LIN {X 0,Y 115.014,Z 337.015,A -85,B 0,C 180,E1 -25713.825,E2 -25713.825} C_VEL
LIN {X 0,Y 114.868,Z 336.176,A -85,B 0,C 180,E1 -25714.155,E2 -25714.155} C_VEL
LIN {X 0,Y 114.957,Z 336.153,A -85,B 0,C 180,E1 -25718.48,E2 -25718.48} C_VEL
LIN {X 0,Y 115.09,Z 336.142,A -85,B 0,C 180,E1 -25725.861,E2 -25725.861} C_VEL
LIN {X 0,Y 115.315,Z 336.105,A -85,B 0,C 180,E1 -25729.464,E2 -25729.464} C_VEL
LIN {X 0,Y 115.522,Z 336.071,A -85,B 0,C 180,E1 -25736.511,E2 -25736.511} C_VEL
LIN {X 0,Y 115.999,Z 336.032,A -85,B 0,C 180,E1 -25739.999,E2 -25739.999} C_VEL
LIN {X 0,Y 115.369,Z 336.065,A -85,B 0,C 180,E1 -25746.997,E2 -25746.997} C_VEL
LIN {X 0,Y 115.214,Z 336.133,A -85,B 0,C 180,E1 -25752.56,E2 -25752.56} C_VEL
LIN {X 0,Y 114.993,Z 336.157,A -85,B 0,C 180,E1 -25757.793,E2 -25757.793} C_VEL
LIN {X 0,Y 114.954,Z 336.155,A -85,B 0,C 180,E1 -25763.488,E2 -25763.488} C_VEL
LIN {X 0,Y 114.864,Z 336.171,A -85,B 0,C 180,E1 -25771.054,E2 -25771.054} C_VEL
LIN {X 0,Y 114.786,Z 336.182,A -85,B 0,C 180,E1 -25777.753,E2 -25777.753} C_VEL
LIN {X 0,Y 114.854,Z 336.215,A -85,B 0,C 180,E1 -25781.569,E2 -25781.569} C_VEL
LIN {X 0,Y 115.591,Z 338.609,A -85,B 0,C 180,E1 -25782.393,E2 -25782.393} C_VEL
LIN {X 0,Y 117.297,Z 340.754,A -85,B 0,C 180,E1 -25783.84,E2 -25783.84} C_VEL
LIN {X 0,Y 118.632,Z 341.83,A -85,B 0,C 180,E1 -25784.849,E2 -25784.849} C_VEL
LIN {X 0,Y 120.483,Z 344.932,A -85,B 0,C 180,E1 -25786.329,E2 -25786.329} C_VEL
LIN {X 0,Y 122.291,Z 346.894,A -85,B 0,C 180,E1 -25787.589,E2 -25787.589} C_VEL
LIN {X 0,Y 128.039,Z 355.27,A -85,B 0,C 180,E1 -25791.345,E2 -25791.345} C_VEL
LIN {X 0,Y 132.282,Z 362.156,A -85,B 0,C 180,E1 -25793.819,E2 -25793.819} C_VEL
LIN {X 0,Y 137.779,Z 372.248,A -85,B 0,C 180,E1 -25796.776,E2 -25796.776} C_VEL
LIN {X 0,Y 142.801,Z 383.272,A -85,B 0,C 180,E1 -25799.292,E2 -25799.292} C_VEL
LIN {X 0,Y 139.384,Z 431.741,A -85,B 0,C 180,E1 -25801.446,E2 -25801.446} C_VEL
LIN {X 0,Y 137.61,Z 444.886,A -85,B 0,C 180,E1 -25802.518,E2 -25802.518} C_VEL
LIN {X 0,Y 135.307,Z 457.913,A -85,B 0,C 180,E1 -25804.21,E2 -25804.21} C_VEL
LIN {X 0,Y 132.086,Z 470.579,A -85,B 0,C 180,E1 -25806.476,E2 -25806.476} C_VEL
LIN {X 0,Y 128.848,Z 481.799,A -85,B 0,C 180,E1 -25809.23,E2 -25809.23} C_VEL
LIN {X 0,Y 125.616,Z 491.287,A -85,B 0,C 180,E1 -25812.226,E2 -25812.226} C_VEL
LIN {X 0,Y 122.323,Z 500.241,A -85,B 0,C 180,E1 -25815.862,E2 -25815.862} C_VEL
LIN {X 0,Y 118.762,Z 509.308,A -85,B 0,C 180,E1 -25820.629,E2 -25820.629} C_VEL
LIN {X 0,Y 116.029,Z 516.6,A -85,B 0,C 180,E1 -25825.653,E2 -25825.653} C_VEL
LIN {X 0,Y 114.373,Z 521.514,A -85,B 0,C 180,E1 -25829.995,E2 -25829.995} C_VEL
LIN {X 0,Y 112.963,Z 526.412,A -85,B 0,C 180,E1 -25835.482,E2 -25835.482} C_VEL
LIN {X 0,Y 112.094,Z 529.991,A -85,B 0,C 180,E1 -25840.836,E2 -25840.836} C_VEL
LIN {X 0,Y 111.893,Z 531.873,A -85,B 0,C 180,E1 -25844.545,E2 -25844.545} C_VEL
LIN {X 0,Y 112.339,Z 533.886,A -85,B 0,C 180,E1 -25850.216,E2 -25850.216} C_VEL
LIN {X 0,Y 113.447,Z 534.9,A -85,B 0,C 180,E1 -25855.693,E2 -25855.693} C_VEL
LIN {X 0,Y 115.8,Z 534.902,A -85,B 0,C 180,E1 -25861.826,E2 -25861.826} C_VEL
LIN {X 0,Y 118.399,Z 534.078,A -85,B 0,C 180,E1 -25866.405,E2 -25866.405} C_VEL
LIN {X 0,Y 122.562,Z 532.001,A -85,B 0,C 180,E1 -25871.803,E2 -25871.803} C_VEL
LIN {X 0,Y 126.828,Z 529.279,A -85,B 0,C 180,E1 -25876.078,E2 -25876.078} C_VEL
LIN {X 0,Y 132.129,Z 525.316,A -85,B 0,C 180,E1 -25880.337,E2 -25880.337} C_VEL
LIN {X 0,Y 138.279,Z 519.935,A -85,B 0,C 180,E1 -25884.401,E2 -25884.401} C_VEL
LIN {X 0,Y 145.281,Z 512.794,A -85,B 0,C 180,E1 -25888.21,E2 -25888.21} C_VEL
LIN {X 0,Y 152.135,Z 504.673,A -85,B 0,C 180,E1 -25891.359,E2 -25891.359} C_VEL
LIN {X 0,Y 158.91,Z 495.272,A -85,B 0,C 180,E1 -25894.011,E2 -25894.011} C_VEL
LIN {X 0,Y 165.11,Z 484.9,A -85,B 0,C 180,E1 -25896.218,E2 -25896.218} C_VEL
LIN {X 0,Y 170.629,Z 473.828,A -85,B 0,C 180,E1 -25897.961,E2 -25897.961} C_VEL
LIN {X 0,Y 175.101,Z 462.431,A -85,B 0,C 180,E1 -25899.328,E2 -25899.328} C_VEL
LIN {X 0,Y 179.002,Z 449.556,A -85,B 0,C 180,E1 -25900.427,E2 -25900.427} C_VEL
LIN {X 0,Y 181.7,Z 436.861,A -85,B 0,C 180,E1 -25901.178,E2 -25901.178} C_VEL
LIN {X 0,Y 183.622,Z 421.119,A -85,B 0,C 180,E1 -25901.708,E2 -25901.708} C_VEL
LIN {X 0,Y 183.896,Z 418.251,A -85,B 0,C 180,E1 -25901.788,E2 -25901.788} C_VEL
LIN {X 0,Y 179.881,Z 410.116,A -85,B 0,C 180,E1 -25905.361,E2 -25905.361} C_VEL
LIN {X 0,Y 175.899,Z 402.879,A -85,B 0,C 180,E1 -25909.643,E2 -25909.643} C_VEL
LIN {X 0,Y 173.679,Z 399.15,A -85,B 0,C 180,E1 -25912.59,E2 -25912.59} C_VEL
LIN {X 0,Y 171.748,Z 395.552,A -85,B 0,C 180,E1 -25915.973,E2 -25915.973} C_VEL
LIN {X 0,Y 169.873,Z 392.584,A -85,B 0,C 180,E1 -25920.642,E2 -25920.642} C_VEL
LIN {X 0,Y 169.52,Z 391.116,A -85,B 0,C 180,E1 -25922.377,E2 -25922.377} C_VEL
LIN {X 0,Y 169.178,Z 391.143,A -85,B 0,C 180,E1 -25930.637,E2 -25930.637} C_VEL
LIN {X 0,Y 169.496,Z 391.694,A -85,B 0,C 180,E1 -25932.335,E2 -25932.335} C_VEL
LIN {X 0,Y 171.097,Z 395.184,A -85,B 0,C 180,E1 -25937.359,E2 -25937.359} C_VEL
LIN {X 0,Y 171.896,Z 396.213,A -85,B 0,C 180,E1 -25938.945,E2 -25938.945} C_VEL
LIN {X 0,Y 174.141,Z 400.931,A -85,B 0,C 180,E1 -25942.76,E2 -25942.76} C_VEL
LIN {X 0,Y 176.288,Z 405.612,A -85,B 0,C 180,E1 -25945.614,E2 -25945.614} C_VEL
LIN {X 0,Y 178.988,Z 412.031,A -85,B 0,C 180,E1 -25948.682,E2 -25948.682} C_VEL
LIN {X 0,Y 181.92,Z 419.645,A -85,B 0,C 180,E1 -25951.582,E2 -25951.582} C_VEL
LIN {X 0,Y 183.373,Z 423.898,A -85,B 0,C 180,E1 -25952.919,E2 -25952.919} C_VEL
LIN {X 0,Y 181.387,Z 441.689,A -85,B 0,C 180,E1 -25953.52,E2 -25953.52} C_VEL
LIN {X 0,Y 178.821,Z 454.037,A -85,B 0,C 180,E1 -25954.137,E2 -25954.137} C_VEL
LIN {X 0,Y 174.995,Z 466.814,A -85,B 0,C 180,E1 -25955.105,E2 -25955.105} C_VEL
LIN {X 0,Y 170.124,Z 478.957,A -85,B 0,C 180,E1 -25956.342,E2 -25956.342} C_VEL
LIN {X 0,Y 164.688,Z 489.87,A -85,B 0,C 180,E1 -25957.87,E2 -25957.87} C_VEL
LIN {X 0,Y 158.183,Z 500.692,A -85,B 0,C 180,E1 -25959.974,E2 -25959.974} C_VEL
LIN {X 0,Y 151.946,Z 509.507,A -85,B 0,C 180,E1 -25962.271,E2 -25962.271} C_VEL
LIN {X 0,Y 144.869,Z 518.154,A -85,B 0,C 180,E1 -25965.303,E2 -25965.303} C_VEL
LIN {X 0,Y 138.224,Z 525.085,A -85,B 0,C 180,E1 -25968.631,E2 -25968.631} C_VEL
LIN {X 0,Y 132.194,Z 530.666,A -85,B 0,C 180,E1 -25972.316,E2 -25972.316} C_VEL
LIN {X 0,Y 126.992,Z 535.081,A -85,B 0,C 180,E1 -25976.404,E2 -25976.404} C_VEL
LIN {X 0,Y 123.881,Z 537.431,A -85,B 0,C 180,E1 -25979.303,E2 -25979.303} C_VEL
LIN {X 0,Y 121.001,Z 539.364,A -85,B 0,C 180,E1 -25982.318,E2 -25982.318} C_VEL
LIN {X 0,Y 118.527,Z 540.877,A -85,B 0,C 180,E1 -25985.483,E2 -25985.483} C_VEL
LIN {X 0,Y 116.404,Z 541.961,A -85,B 0,C 180,E1 -25988.767,E2 -25988.767} C_VEL
LIN {X 0,Y 113.635,Z 543.009,A -85,B 0,C 180,E1 -25995.683,E2 -25995.683} C_VEL
LIN {X 0,Y 112.838,Z 542.97,A -85,B 0,C 180,E1 -25999.236,E2 -25999.236} C_VEL
LIN {X 0,Y 112.422,Z 542.512,A -85,B 0,C 180,E1 -26002.823,E2 -26002.823} C_VEL
LIN {X 0,Y 112.337,Z 541.661,A -85,B 0,C 180,E1 -26006.419,E2 -26006.419} C_VEL
LIN {X 0,Y 112.45,Z 540.411,A -85,B 0,C 180,E1 -26010.005,E2 -26010.005} C_VEL
LIN {X 0,Y 112.324,Z 537.663,A -85,B 0,C 180,E1 -26015.391,E2 -26015.391} C_VEL
LIN {X 0,Y 112.812,Z 533.857,A -85,B 0,C 180,E1 -26020.777,E2 -26020.777} C_VEL
LIN {X 0,Y 113.958,Z 528.881,A -85,B 0,C 180,E1 -26026.118,E2 -26026.118} C_VEL
LIN {X 0,Y 116.11,Z 522.613,A -85,B 0,C 180,E1 -26031.3,E2 -26031.3} C_VEL
LIN {X 0,Y 119.023,Z 514.744,A -85,B 0,C 180,E1 -26036.291,E2 -26036.291} C_VEL
LIN {X 0,Y 121.441,Z 508.027,A -85,B 0,C 180,E1 -26039.69,E2 -26039.69} C_VEL
LIN {X 0,Y 124.527,Z 500.023,A -85,B 0,C 180,E1 -26042.908,E2 -26042.908} C_VEL
LIN {X 0,Y 127.974,Z 489.74,A -85,B 0,C 180,E1 -26046.188,E2 -26046.188} C_VEL
LIN {X 0,Y 128.825,Z 487.057,A -85,B 0,C 180,E1 -26046.906,E2 -26046.906} C_VEL
LIN {X 0,Y 130.77,Z 488.171,A -85,B 0,C 180,E1 -26048.275,E2 -26048.275} C_VEL
LIN {X 0,Y 130.77,Z 550.146,A -85,B 0,C 180,E1 -26048.275,E2 -26048.275} C_VEL
LIN {X 0,Y 112.288,Z 550.146,A -85,B 0,C 180,E1 -26012.241,E2 -26012.241} C_VEL
LIN {X 0,Y 112.475,Z 548.146,A -85,B 0,C 180,E1 -26011.226,E2 -26011.226} C_VEL
LIN {X 0,Y 112.475,Z 542.371,A -85,B 0,C 180,E1 -26011.226,E2 -26011.226} C_VEL
LIN {X 0,Y 112.45,Z 540.411,A -85,B 0,C 180,E1 -26010.005,E2 -26010.005} C_VEL
LIN {X 0,Y 111.781,Z 539.072,A -85,B 0,C 180,E1 -26012.92,E2 -26012.92} C_VEL
LIN {X 0,Y 110.239,Z 537.452,A -85,B 0,C 180,E1 -26015.767,E2 -26015.767} C_VEL
LIN {X 0,Y 106.959,Z 533.382,A -85,B 0,C 180,E1 -26021.49,E2 -26021.49} C_VEL
LIN {X 0,Y 106.435,Z 530.884,A -85,B 0,C 180,E1 -26024.401,E2 -26024.401} C_VEL
LIN {X 0,Y 106.583,Z 529.982,A -85,B 0,C 180,E1 -26025.356,E2 -26025.356} C_VEL
LIN {X 0,Y 109.008,Z 522.962,A -85,B 0,C 180,E1 -26031.765,E2 -26031.765} C_VEL
LIN {X 0,Y 112.033,Z 515.278,A -85,B 0,C 180,E1 -26037.058,E2 -26037.058} C_VEL
LIN {X 0,Y 114.607,Z 508.534,A -85,B 0,C 180,E1 -26040.709,E2 -26040.709} C_VEL
LIN {X 0,Y 118.178,Z 499.845,A -85,B 0,C 180,E1 -26044.405,E2 -26044.405} C_VEL
LIN {X 0,Y 121.825,Z 489.591,A -85,B 0,C 180,E1 -26047.809,E2 -26047.809} C_VEL
LIN {X 0,Y 125.604,Z 478.233,A -85,B 0,C 180,E1 -26050.582,E2 -26050.582} C_VEL
LIN {X 0,Y 128.836,Z 466.435,A -85,B 0,C 180,E1 -26052.73,E2 -26052.73} C_VEL
LIN {X 0,Y 131.586,Z 453.372,A -85,B 0,C 180,E1 -26054.409,E2 -26054.409} C_VEL
LIN {X 0,Y 133.537,Z 440.115,A -85,B 0,C 180,E1 -26055.511,E2 -26055.511} C_VEL
LIN {X 0,Y 136.289,Z 402.278,A -85,B 0,C 180,E1 -26057.286,E2 -26057.286} C_VEL
LIN {X 0,Y 136.391,Z 396.466,A -85,B 0,C 180,E1 -26057.652,E2 -26057.652} C_VEL
LIN {X 0,Y 135.806,Z 387.938,A -85,B 0,C 180,E1 -26058.466,E2 -26058.466} C_VEL
LIN {X 0,Y 132.059,Z 376.712,A -85,B 0,C 180,E1 -26060.773,E2 -26060.773} C_VEL
LIN {X 0,Y 127.862,Z 366.383,A -85,B 0,C 180,E1 -26063.444,E2 -26063.444} C_VEL
LIN {X 0,Y 122.784,Z 358.228,A -85,B 0,C 180,E1 -26066.707,E2 -26066.707} C_VEL
LIN {X 0,Y 120.388,Z 354.639,A -85,B 0,C 180,E1 -26068.403,E2 -26068.403} C_VEL
LIN {X 0,Y 118.264,Z 351.547,A -85,B 0,C 180,E1 -26070.012,E2 -26070.012} C_VEL
LIN {X 0,Y 115.776,Z 347.918,A -85,B 0,C 180,E1 -26072.059,E2 -26072.059} C_VEL
LIN {X 0,Y 112.849,Z 344.495,A -85,B 0,C 180,E1 -26074.634,E2 -26074.634} C_VEL
LIN {X 0,Y 111.991,Z 342.667,A -85,B 0,C 180,E1 -26075.552,E2 -26075.552} C_VEL
LIN {X 0,Y 109.423,Z 340.621,A -85,B 0,C 180,E1 -26078.078,E2 -26078.078} C_VEL
LIN {X 0,Y 108.124,Z 338.229,A -85,B 0,C 180,E1 -26079.674,E2 -26079.674} C_VEL
LIN {X 0,Y 107.884,Z 337.013,A -85,B 0,C 180,E1 -26080.248,E2 -26080.248} C_VEL
LIN {X 0,Y 108.233,Z 336.994,A -85,B 0,C 180,E1 -26088.766,E2 -26088.766} C_VEL
LIN {X 0,Y 108.445,Z 336.947,A -85,B 0,C 180,E1 -26096.283,E2 -26096.283} C_VEL
LIN {X 0,Y 108.949,Z 336.91,A -85,B 0,C 180,E1 -26099.999,E2 -26099.999} C_VEL
LIN {X 0,Y 108.307,Z 336.945,A -85,B 0,C 180,E1 -26107.456,E2 -26107.456} C_VEL
LIN {X 0,Y 108.148,Z 337.012,A -85,B 0,C 180,E1 -26112.875,E2 -26112.875} C_VEL
LIN {X 0,Y 107.893,Z 337.046,A -85,B 0,C 180,E1 -26119.007,E2 -26119.007} C_VEL
LIN {X 0,Y 107.863,Z 337.042,A -85,B 0,C 180,E1 -26124.178,E2 -26124.178} C_VEL
LIN {X 0,Y 107.787,Z 337.055,A -85,B 0,C 180,E1 -26132.036,E2 -26132.036} C_VEL
LIN {X 0,Y 107.714,Z 337.052,A -85,B 0,C 180,E1 -26135.282,E2 -26135.282} C_VEL
LIN {X 0,Y 108.497,Z 339.503,A -85,B 0,C 180,E1 -26136.472,E2 -26136.472} C_VEL
LIN {X 0,Y 110.46,Z 341.809,A -85,B 0,C 180,E1 -26138.628,E2 -26138.628} C_VEL
LIN {X 0,Y 112.058,Z 343.005,A -85,B 0,C 180,E1 -26140.151,E2 -26140.151} C_VEL
LIN {X 0,Y 113.914,Z 346.117,A -85,B 0,C 180,E1 -26141.99,E2 -26141.99} C_VEL
LIN {X 0,Y 115.783,Z 348.108,A -85,B 0,C 180,E1 -26143.577,E2 -26143.577} C_VEL
LIN {X 0,Y 118.166,Z 351.553,A -85,B 0,C 180,E1 -26145.537,E2 -26145.537} C_VEL
LIN {X 0,Y 119.657,Z 353.54,A -85,B 0,C 180,E1 -26146.664,E2 -26146.664} C_VEL
LIN {X 0,Y 122.74,Z 358.12,A -85,B 0,C 180,E1 -26148.87,E2 -26148.87} C_VEL
LIN {X 0,Y 127.329,Z 365.315,A -85,B 0,C 180,E1 -26151.83,E2 -26151.83} C_VEL
LIN {X 0,Y 133.258,Z 376.523,A -85,B 0,C 180,E1 -26155.313,E2 -26155.313} C_VEL
LIN {X 0,Y 137.199,Z 385.403,A -85,B 0,C 180,E1 -26157.479,E2 -26157.479} C_VEL
LIN {X 0,Y 133.843,Z 431.591,A -85,B 0,C 180,E1 -26159.582,E2 -26159.582} C_VEL
LIN {X 0,Y 131.946,Z 445.124,A -85,B 0,C 180,E1 -26160.701,E2 -26160.701} C_VEL
LIN {X 0,Y 129.644,Z 457.561,A -85,B 0,C 180,E1 -26162.338,E2 -26162.338} C_VEL
LIN {X 0,Y 126.52,Z 469.574,A -85,B 0,C 180,E1 -26164.496,E2 -26164.496} C_VEL
LIN {X 0,Y 123.024,Z 481.038,A -85,B 0,C 180,E1 -26167.314,E2 -26167.314} C_VEL
LIN {X 0,Y 119.246,Z 491.703,A -85,B 0,C 180,E1 -26170.771,E2 -26170.771} C_VEL
LIN {X 0,Y 115.43,Z 501.491,A -85,B 0,C 180,E1 -26174.998,E2 -26174.998} C_VEL
LIN {X 0,Y 111.728,Z 510.395,A -85,B 0,C 180,E1 -26180.033,E2 -26180.033} C_VEL
LIN {X 0,Y 108.909,Z 517.496,A -85,B 0,C 180,E1 -26185.368,E2 -26185.368} C_VEL
LIN {X 0,Y 106.664,Z 523.991,A -85,B 0,C 180,E1 -26191.882,E2 -26191.882} C_VEL
LIN {X 0,Y 105.388,Z 528.295,A -85,B 0,C 180,E1 -26197.659,E2 -26197.659} C_VEL
LIN {X 0,Y 104.909,Z 530.585,A -85,B 0,C 180,E1 -26201.588,E2 -26201.588} C_VEL
LIN {X 0,Y 104.832,Z 532.37,A -85,B 0,C 180,E1 -26205.549,E2 -26205.549} C_VEL
LIN {X 0,Y 105.315,Z 534.131,A -85,B 0,C 180,E1 -26210.893,E2 -26210.893} C_VEL
LIN {X 0,Y 106.784,Z 535.206,A -85,B 0,C 180,E1 -26217.426,E2 -26217.426} C_VEL
LIN {X 0,Y 109.182,Z 535.186,A -85,B 0,C 180,E1 -26223.197,E2 -26223.197} C_VEL
LIN {X 0,Y 112.465,Z 534.206,A -85,B 0,C 180,E1 -26228.668,E2 -26228.668} C_VEL
LIN {X 0,Y 116.503,Z 532.329,A -85,B 0,C 180,E1 -26233.624,E2 -26233.624} C_VEL
LIN {X 0,Y 121.744,Z 529.197,A -85,B 0,C 180,E1 -26238.622,E2 -26238.622} C_VEL
LIN {X 0,Y 127.935,Z 524.741,A -85,B 0,C 180,E1 -26243.248,E2 -26243.248} C_VEL
LIN {X 0,Y 135.24,Z 518.552,A -85,B 0,C 180,E1 -26247.605,E2 -26247.605} C_VEL
LIN {X 0,Y 142.361,Z 511.408,A -85,B 0,C 180,E1 -26251.185,E2 -26251.185} C_VEL
LIN {X 0,Y 148.709,Z 504.022,A -85,B 0,C 180,E1 -26253.878,E2 -26253.878} C_VEL
LIN {X 0,Y 156.056,Z 493.977,A -85,B 0,C 180,E1 -26256.565,E2 -26256.565} C_VEL
LIN {X 0,Y 162.272,Z 483.769,A -85,B 0,C 180,E1 -26258.605,E2 -26258.605} C_VEL
LIN {X 0,Y 167.844,Z 472.54,A -85,B 0,C 180,E1 -26260.271,E2 -26260.271} C_VEL
LIN {X 0,Y 172.183,Z 461.515,A -85,B 0,C 180,E1 -26261.532,E2 -26261.532} C_VEL
LIN {X 0,Y 176.081,Z 448.852,A -85,B 0,C 180,E1 -26262.54,E2 -26262.54} C_VEL
LIN {X 0,Y 178.754,Z 436.204,A -85,B 0,C 180,E1 -26263.234,E2 -26263.234} C_VEL
LIN {X 0,Y 180.477,Z 421.837,A -85,B 0,C 180,E1 -26263.747,E2 -26263.747} C_VEL
LIN {X 0,Y 177.478,Z 415.559,A -85,B 0,C 180,E1 -26266.693,E2 -26266.693} C_VEL
LIN {X 0,Y 174.264,Z 409.34,A -85,B 0,C 180,E1 -26270.44,E2 -26270.44} C_VEL
LIN {X 0,Y 172.165,Z 405.604,A -85,B 0,C 180,E1 -26273.463,E2 -26273.463} C_VEL
LIN {X 0,Y 170.378,Z 402.196,A -85,B 0,C 180,E1 -26276.868,E2 -26276.868} C_VEL
LIN {X 0,Y 168.764,Z 399.205,A -85,B 0,C 180,E1 -26281.47,E2 -26281.47} C_VEL
LIN {X 0,Y 168.5,Z 398.13,A -85,B 0,C 180,E1 -26282.935,E2 -26282.935} C_VEL
LIN {X 0,Y 168.304,Z 398.198,A -85,B 0,C 180,E1 -26290.693,E2 -26290.693} C_VEL
LIN {X 0,Y 168.561,Z 398.894,A -85,B 0,C 180,E1 -26292.219,E2 -26292.219} C_VEL
LIN {X 0,Y 170.088,Z 402.194,A -85,B 0,C 180,E1 -26297.139,E2 -26297.139} C_VEL
LIN {X 0,Y 170.73,Z 403.147,A -85,B 0,C 180,E1 -26298.49,E2 -26298.49} C_VEL
LIN {X 0,Y 172.617,Z 407.458,A -85,B 0,C 180,E1 -26301.967,E2 -26301.967} C_VEL
LIN {X 0,Y 174.622,Z 412.185,A -85,B 0,C 180,E1 -26304.84,E2 -26304.84} C_VEL
LIN {X 0,Y 176.985,Z 418.269,A -85,B 0,C 180,E1 -26307.734,E2 -26307.734} C_VEL
LIN {X 0,Y 179.551,Z 425.417,A -85,B 0,C 180,E1 -26310.48,E2 -26310.48} C_VEL
LIN {X 0,Y 180.048,Z 426.922,A -85,B 0,C 180,E1 -26310.982,E2 -26310.982} C_VEL
LIN {X 0,Y 178.187,Z 442.271,A -85,B 0,C 180,E1 -26311.515,E2 -26311.515} C_VEL
LIN {X 0,Y 175.536,Z 454.311,A -85,B 0,C 180,E1 -26312.107,E2 -26312.107} C_VEL
LIN {X 0,Y 171.781,Z 466.448,A -85,B 0,C 180,E1 -26313.004,E2 -26313.004} C_VEL
LIN {X 0,Y 166.764,Z 478.644,A -85,B 0,C 180,E1 -26314.209,E2 -26314.209} C_VEL
LIN {X 0,Y 161.155,Z 489.569,A -85,B 0,C 180,E1 -26315.692,E2 -26315.692} C_VEL
LIN {X 0,Y 155.025,Z 499.437,A -85,B 0,C 180,E1 -26317.507,E2 -26317.507} C_VEL
LIN {X 0,Y 148.578,Z 508.406,A -85,B 0,C 180,E1 -26319.774,E2 -26319.774} C_VEL
LIN {X 0,Y 141.125,Z 517.196,A -85,B 0,C 180,E1 -26322.738,E2 -26322.738} C_VEL
LIN {X 0,Y 134.129,Z 524.28,A -85,B 0,C 180,E1 -26326.038,E2 -26326.038} C_VEL
LIN {X 0,Y 128.649,Z 529.093,A -85,B 0,C 180,E1 -26329.045,E2 -26329.045} C_VEL
LIN {X 0,Y 122.167,Z 534.331,A -85,B 0,C 180,E1 -26333.649,E2 -26333.649} C_VEL
LIN {X 0,Y 117.829,Z 537.408,A -85,B 0,C 180,E1 -26337.54,E2 -26337.54} C_VEL
LIN {X 0,Y 114.739,Z 539.298,A -85,B 0,C 180,E1 -26340.665,E2 -26340.665} C_VEL
LIN {X 0,Y 109.8,Z 541.787,A -85,B 0,C 180,E1 -26347.422,E2 -26347.422} C_VEL
LIN {X 0,Y 106.742,Z 542.762,A -85,B 0,C 180,E1 -26354.736,E2 -26354.736} C_VEL
LIN {X 0,Y 105.846,Z 542.66,A -85,B 0,C 180,E1 -26358.516,E2 -26358.516} C_VEL
LIN {X 0,Y 105.247,Z 541.267,A -85,B 0,C 180,E1 -26366.177,E2 -26366.177} C_VEL
LIN {X 0,Y 105.363,Z 539.981,A -85,B 0,C 180,E1 -26370.006,E2 -26370.006} C_VEL
LIN {X 0,Y 105.246,Z 537.154,A -85,B 0,C 180,E1 -26375.754,E2 -26375.754} C_VEL
LIN {X 0,Y 105.819,Z 533.265,A -85,B 0,C 180,E1 -26381.498,E2 -26381.498} C_VEL
LIN {X 0,Y 106.583,Z 529.982,A -85,B 0,C 180,E1 -26385.356,E2 -26385.356} C_VEL
LIN {X 0,Y 106.777,Z 527.242,A -85,B 0,C 180,E1 -26388.149,E2 -26388.149} C_VEL
LIN {X 0,Y 105.462,Z 520.11,A -85,B 0,C 180,E1 -26394.559,E2 -26394.559} C_VEL
LIN {X 0,Y 105.55,Z 515.464,A -85,B 0,C 180,E1 -26398.057,E2 -26398.057} C_VEL
LIN {X 0,Y 106.301,Z 512.936,A -85,B 0,C 180,E1 -26399.661,E2 -26399.661} C_VEL
LIN {X 0,Y 108.392,Z 507.863,A -85,B 0,C 180,E1 -26402.453,E2 -26402.453} C_VEL
LIN {X 0,Y 111.922,Z 499.669,A -85,B 0,C 180,E1 -26406.07,E2 -26406.07} C_VEL
LIN {X 0,Y 115.783,Z 489.442,A -85,B 0,C 180,E1 -26409.601,E2 -26409.601} C_VEL
LIN {X 0,Y 119.757,Z 478.111,A -85,B 0,C 180,E1 -26412.451,E2 -26412.451} C_VEL
LIN {X 0,Y 123.145,Z 466.349,A -85,B 0,C 180,E1 -26414.649,E2 -26414.649} C_VEL
LIN {X 0,Y 125.989,Z 453.545,A -85,B 0,C 180,E1 -26416.345,E2 -26416.345} C_VEL
LIN {X 0,Y 128.06,Z 440.152,A -85,B 0,C 180,E1 -26417.49,E2 -26417.49} C_VEL
LIN {X 0,Y 130.485,Z 409.714,A -85,B 0,C 180,E1 -26418.949,E2 -26418.949} C_VEL
LIN {X 0,Y 131.097,Z 397.951,A -85,B 0,C 180,E1 -26419.577,E2 -26419.577} C_VEL
LIN {X 0,Y 130.616,Z 390.316,A -85,B 0,C 180,E1 -26420.348,E2 -26420.348} C_VEL
LIN {X 0,Y 126.989,Z 379.052,A -85,B 0,C 180,E1 -26422.825,E2 -26422.825} C_VEL
LIN {X 0,Y 123.314,Z 370.227,A -85,B 0,C 180,E1 -26425.362,E2 -26425.362} C_VEL
LIN {X 0,Y 118.846,Z 362.746,A -85,B 0,C 180,E1 -26428.547,E2 -26428.547} C_VEL
LIN {X 0,Y 115.21,Z 357.304,A -85,B 0,C 180,E1 -26431.444,E2 -26431.444} C_VEL
LIN {X 0,Y 112.321,Z 353.2,A -85,B 0,C 180,E1 -26434.023,E2 -26434.023} C_VEL
LIN {X 0,Y 109.698,Z 349.548,A -85,B 0,C 180,E1 -26436.651,E2 -26436.651} C_VEL
LIN {X 0,Y 109.131,Z 348.721,A -85,B 0,C 180,E1 -26437.269,E2 -26437.269} C_VEL
LIN {X 0,Y 106.68,Z 346.151,A -85,B 0,C 180,E1 -26440.016,E2 -26440.016} C_VEL
LIN {X 0,Y 105.401,Z 343.672,A -85,B 0,C 180,E1 -26441.786,E2 -26441.786} C_VEL
LIN {X 0,Y 102.983,Z 342.054,A -85,B 0,C 180,E1 -26445.041,E2 -26445.041} C_VEL
LIN {X 0,Y 101.591,Z 339.692,A -85,B 0,C 180,E1 -26447.497,E2 -26447.497} C_VEL
LIN {X 0,Y 101.195,Z 337.869,A -85,B 0,C 180,E1 -26448.735,E2 -26448.735} C_VEL
LIN {X 0,Y 101.367,Z 337.823,A -85,B 0,C 180,E1 -26456.023,E2 -26456.023} C_VEL
LIN {X 0,Y 101.872,Z 337.791,A -85,B 0,C 180,E1 -26459.999,E2 -26459.999} C_VEL
LIN {X 0,Y 101.242,Z 337.827,A -85,B 0,C 180,E1 -26467.98,E2 -26467.98} C_VEL
LIN {X 0,Y 101.063,Z 337.894,A -85,B 0,C 180,E1 -26473.18,E2 -26473.18} C_VEL
LIN {X 0,Y 100.812,Z 337.922,A -85,B 0,C 180,E1 -26480.399,E2 -26480.399} C_VEL
LIN {X 0,Y 100.737,Z 337.938,A -85,B 0,C 180,E1 -26486.35,E2 -26486.35} C_VEL
LIN {X 0,Y 101.381,Z 340.194,A -85,B 0,C 180,E1 -26487.898,E2 -26487.898} C_VEL
LIN {X 0,Y 102.916,Z 342.262,A -85,B 0,C 180,E1 -26490.523,E2 -26490.523} C_VEL
LIN {X 0,Y 105.418,Z 343.993,A -85,B 0,C 180,E1 -26493.887,E2 -26493.887} C_VEL
LIN {X 0,Y 107.138,Z 347.037,A -85,B 0,C 180,E1 -26496.183,E2 -26496.183} C_VEL
LIN {X 0,Y 109.505,Z 349.285,A -85,B 0,C 180,E1 -26498.748,E2 -26498.748} C_VEL
LIN {X 0,Y 111.832,Z 352.759,A -85,B 0,C 180,E1 -26501.147,E2 -26501.147} C_VEL
LIN {X 0,Y 113.125,Z 354.404,A -85,B 0,C 180,E1 -26502.34,E2 -26502.34} C_VEL
LIN {X 0,Y 116.778,Z 359.649,A -85,B 0,C 180,E1 -26505.46,E2 -26505.46} C_VEL
LIN {X 0,Y 121.44,Z 366.898,A -85,B 0,C 180,E1 -26508.948,E2 -26508.948} C_VEL
LIN {X 0,Y 125.323,Z 373.822,A -85,B 0,C 180,E1 -26511.566,E2 -26511.566} C_VEL
LIN {X 0,Y 129.773,Z 382.848,A -85,B 0,C 180,E1 -26514.324,E2 -26514.324} C_VEL
LIN {X 0,Y 131.798,Z 387.458,A -85,B 0,C 180,E1 -26515.529,E2 -26515.529} C_VEL
LIN {X 0,Y 128.449,Z 431.58,A -85,B 0,C 180,E1 -26517.573,E2 -26517.573} C_VEL
LIN {X 0,Y 126.557,Z 444.739,A -85,B 0,C 180,E1 -26518.666,E2 -26518.666} C_VEL
LIN {X 0,Y 124.132,Z 457.17,A -85,B 0,C 180,E1 -26520.299,E2 -26520.299} C_VEL
LIN {X 0,Y 121.125,Z 468.561,A -85,B 0,C 180,E1 -26522.338,E2 -26522.338} C_VEL
LIN {X 0,Y 117.786,Z 478.986,A -85,B 0,C 180,E1 -26524.836,E2 -26524.836} C_VEL
LIN {X 0,Y 114.308,Z 488.648,A -85,B 0,C 180,E1 -26527.872,E2 -26527.872} C_VEL
LIN {X 0,Y 110.729,Z 497.609,A -85,B 0,C 180,E1 -26531.492,E2 -26531.492} C_VEL
LIN {X 0,Y 107.17,Z 505.849,A -85,B 0,C 180,E1 -26535.758,E2 -26535.758} C_VEL
LIN {X 0,Y 103.62,Z 513.934,A -85,B 0,C 180,E1 -26541.216,E2 -26541.216} C_VEL
LIN {X 0,Y 101.392,Z 519.395,A -85,B 0,C 180,E1 -26546.019,E2 -26546.019} C_VEL
LIN {X 0,Y 99.472,Z 524.753,A -85,B 0,C 180,E1 -26552.018,E2 -26552.018} C_VEL
LIN {X 0,Y 98.188,Z 528.949,A -85,B 0,C 180,E1 -26558.224,E2 -26558.224} C_VEL
LIN {X 0,Y 97.771,Z 531.138,A -85,B 0,C 180,E1 -26562.447,E2 -26562.447} C_VEL
LIN {X 0,Y 97.78,Z 532.87,A -85,B 0,C 180,E1 -26566.702,E2 -26566.702} C_VEL
LIN {X 0,Y 98.316,Z 534.376,A -85,B 0,C 180,E1 -26571.678,E2 -26571.678} C_VEL
LIN {X 0,Y 100.229,Z 535.509,A -85,B 0,C 180,E1 -26579.388,E2 -26579.388} C_VEL
LIN {X 0,Y 102.616,Z 535.473,A -85,B 0,C 180,E1 -26584.73,E2 -26584.73} C_VEL
LIN {X 0,Y 106.722,Z 534.309,A -85,B 0,C 180,E1 -26591.18,E2 -26591.18} C_VEL
LIN {X 0,Y 110.62,Z 532.649,A -85,B 0,C 180,E1 -26595.665,E2 -26595.665} C_VEL
LIN {X 0,Y 116.941,Z 529.1,A -85,B 0,C 180,E1 -26601.369,E2 -26601.369} C_VEL
LIN {X 0,Y 123.24,Z 524.822,A -85,B 0,C 180,E1 -26605.768,E2 -26605.768} C_VEL
LIN {X 0,Y 130.179,Z 519.259,A -85,B 0,C 180,E1 -26609.735,E2 -26609.735} C_VEL
LIN {X 0,Y 137.627,Z 512.223,A -85,B 0,C 180,E1 -26613.324,E2 -26613.324} C_VEL
LIN {X 0,Y 144.238,Z 504.975,A -85,B 0,C 180,E1 -26615.995,E2 -26615.995} C_VEL
LIN {X 0,Y 151.157,Z 496.121,A -85,B 0,C 180,E1 -26618.406,E2 -26618.406} C_VEL
LIN {X 0,Y 157.534,Z 486.288,A -85,B 0,C 180,E1 -26620.453,E2 -26620.453} C_VEL
LIN {X 0,Y 163.36,Z 475.538,A -85,B 0,C 180,E1 -26622.097,E2 -26622.097} C_VEL
LIN {X 0,Y 168.547,Z 463.375,A -85,B 0,C 180,E1 -26623.53,E2 -26623.53} C_VEL
LIN {X 0,Y 172.708,Z 450.629,A -85,B 0,C 180,E1 -26624.553,E2 -26624.553} C_VEL
LIN {X 0,Y 175.707,Z 437.47,A -85,B 0,C 180,E1 -26625.296,E2 -26625.296} C_VEL
LIN {X 0,Y 177.311,Z 425.616,A -85,B 0,C 180,E1 -26625.731,E2 -26625.731} C_VEL
LIN {X 0,Y 174.815,Z 420.287,A -85,B 0,C 180,E1 -26628.478,E2 -26628.478} C_VEL
LIN {X 0,Y 172.076,Z 414.755,A -85,B 0,C 180,E1 -26632.079,E2 -26632.079} C_VEL
LIN {X 0,Y 170.469,Z 411.666,A -85,B 0,C 180,E1 -26634.752,E2 -26634.752} C_VEL
LIN {X 0,Y 169.238,Z 409.053,A -85,B 0,C 180,E1 -26637.363,E2 -26637.363} C_VEL
LIN {X 0,Y 167.74,Z 406.035,A -85,B 0,C 180,E1 -26642.03,E2 -26642.03} C_VEL
LIN {X 0,Y 167.595,Z 405.215,A -85,B 0,C 180,E1 -26643.005,E2 -26643.005} C_VEL
LIN {X 0,Y 167.271,Z 405.14,A -85,B 0,C 180,E1 -26649.676,E2 -26649.676} C_VEL
LIN {X 0,Y 167.534,Z 405.524,A -85,B 0,C 180,E1 -26651.424,E2 -26651.424} C_VEL
LIN {X 0,Y 168.977,Z 409.056,A -85,B 0,C 180,E1 -26656.671,E2 -26656.671} C_VEL
LIN {X 0,Y 169.543,Z 410.024,A -85,B 0,C 180,E1 -26657.961,E2 -26657.961} C_VEL
LIN {X 0,Y 171.212,Z 414.187,A -85,B 0,C 180,E1 -26661.286,E2 -26661.286} C_VEL
LIN {X 0,Y 172.786,Z 418.25,A -85,B 0,C 180,E1 -26663.762,E2 -26663.762} C_VEL
LIN {X 0,Y 174.983,Z 424.338,A -85,B 0,C 180,E1 -26666.702,E2 -26666.702} C_VEL
LIN {X 0,Y 176.896,Z 430.069,A -85,B 0,C 180,E1 -26668.954,E2 -26668.954} C_VEL
LIN {X 0,Y 175.162,Z 443.005,A -85,B 0,C 180,E1 -26669.439,E2 -26669.439} C_VEL
LIN {X 0,Y 172.277,Z 455.274,A -85,B 0,C 180,E1 -26670.05,E2 -26670.05} C_VEL
LIN {X 0,Y 168.043,Z 468.1,A -85,B 0,C 180,E1 -26670.986,E2 -26670.986} C_VEL
LIN {X 0,Y 162.901,Z 479.873,A -85,B 0,C 180,E1 -26672.156,E2 -26672.156} C_VEL
LIN {X 0,Y 157.15,Z 490.441,A -85,B 0,C 180,E1 -26673.606,E2 -26673.606} C_VEL
LIN {X 0,Y 150.831,Z 500.115,A -85,B 0,C 180,E1 -26675.379,E2 -26675.379} C_VEL
LIN {X 0,Y 144.159,Z 508.929,A -85,B 0,C 180,E1 -26677.615,E2 -26677.615} C_VEL
LIN {X 0,Y 136.426,Z 517.576,A -85,B 0,C 180,E1 -26680.557,E2 -26680.557} C_VEL
LIN {X 0,Y 129.129,Z 524.506,A -85,B 0,C 180,E1 -26683.858,E2 -26683.858} C_VEL
LIN {X 0,Y 123.368,Z 529.266,A -85,B 0,C 180,E1 -26686.881,E2 -26686.881} C_VEL
LIN {X 0,Y 115.983,Z 534.712,A -85,B 0,C 180,E1 -26691.975,E2 -26691.975} C_VEL
LIN {X 0,Y 111.9,Z 537.395,A -85,B 0,C 180,E1 -26695.587,E2 -26695.587} C_VEL
LIN {X 0,Y 108.589,Z 539.213,A -85,B 0,C 180,E1 -26698.824,E2 -26698.824} C_VEL
LIN {X 0,Y 103.269,Z 541.613,A -85,B 0,C 180,E1 -26705.907,E2 -26705.907} C_VEL
LIN {X 0,Y 99.87,Z 542.502,A -85,B 0,C 180,E1 -26713.658,E2 -26713.658} C_VEL
LIN {X 0,Y 98.309,Z 541.797,A -85,B 0,C 180,E1 -26721.786,E2 -26721.786} C_VEL
LIN {X 0,Y 98.166,Z 540.874,A -85,B 0,C 180,E1 -26725.901,E2 -26725.901} C_VEL
LIN {X 0,Y 98.277,Z 539.549,A -85,B 0,C 180,E1 -26730.006,E2 -26730.006} C_VEL
LIN {X 0,Y 98.192,Z 536.647,A -85,B 0,C 180,E1 -26736.169,E2 -26736.169} C_VEL
LIN {X 0,Y 98.823,Z 532.671,A -85,B 0,C 180,E1 -26742.325,E2 -26742.325} C_VEL
LIN {X 0,Y 100.624,Z 526.498,A -85,B 0,C 180,E1 -26749.382,E2 -26749.382} C_VEL
LIN {X 0,Y 103.404,Z 519.745,A -85,B 0,C 180,E1 -26755.143,E2 -26755.143} C_VEL
LIN {X 0,Y 106.301,Z 512.936,A -85,B 0,C 180,E1 -26759.661,E2 -26759.661} C_VEL
LIN {X 0,Y 107.342,Z 509.037,A -85,B 0,C 180,E1 -26761.979,E2 -26761.979} C_VEL
LIN {X 0,Y 107.694,Z 502.306,A -85,B 0,C 180,E1 -26765.857,E2 -26765.857} C_VEL
LIN {X 0,Y 108.223,Z 495.073,A -85,B 0,C 180,E1 -26769.454,E2 -26769.454} C_VEL
LIN {X 0,Y 109.465,Z 490.38,A -85,B 0,C 180,E1 -26771.237,E2 -26771.237} C_VEL
LIN {X 0,Y 113.486,Z 479.576,A -85,B 0,C 180,E1 -26774.169,E2 -26774.169} C_VEL
LIN {X 0,Y 117.309,Z 467.259,A -85,B 0,C 180,E1 -26776.593,E2 -26776.593} C_VEL
LIN {X 0,Y 120.445,Z 454.303,A -85,B 0,C 180,E1 -26778.391,E2 -26778.391} C_VEL
LIN {X 0,Y 122.641,Z 441.193,A -85,B 0,C 180,E1 -26779.566,E2 -26779.566} C_VEL
LIN {X 0,Y 124.346,Z 422.73,A -85,B 0,C 180,E1 -26780.518,E2 -26780.518} C_VEL
LIN {X 0,Y 125.942,Z 399.127,A -85,B 0,C 180,E1 -26781.69,E2 -26781.69} C_VEL
LIN {X 0,Y 125.616,Z 392.77,A -85,B 0,C 180,E1 -26782.349,E2 -26782.349} C_VEL
LIN {X 0,Y 122.351,Z 382.415,A -85,B 0,C 180,E1 -26784.799,E2 -26784.799} C_VEL
LIN {X 0,Y 119.433,Z 375.041,A -85,B 0,C 180,E1 -26787.037,E2 -26787.037} C_VEL
LIN {X 0,Y 114.828,Z 366.975,A -85,B 0,C 180,E1 -26790.682,E2 -26790.682} C_VEL
LIN {X 0,Y 111.464,Z 361.968,A -85,B 0,C 180,E1 -26793.667,E2 -26793.667} C_VEL
LIN {X 0,Y 109.426,Z 358.927,A -85,B 0,C 180,E1 -26795.692,E2 -26795.692} C_VEL
LIN {X 0,Y 106.653,Z 354.888,A -85,B 0,C 180,E1 -26798.781,E2 -26798.781} C_VEL
LIN {X 0,Y 104.227,Z 351.912,A -85,B 0,C 180,E1 -26801.828,E2 -26801.828} C_VEL
LIN {X 0,Y 103.306,Z 350.243,A -85,B 0,C 180,E1 -26803.193,E2 -26803.193} C_VEL
LIN {X 0,Y 100.918,Z 348.191,A -85,B 0,C 180,E1 -26806.784,E2 -26806.784} C_VEL
LIN {X 0,Y 99.562,Z 345.436,A -85,B 0,C 180,E1 -26809.578,E2 -26809.578} C_VEL
LIN {X 0,Y 99.253,Z 344.686,A -85,B 0,C 180,E1 -26810.318,E2 -26810.318} C_VEL
LIN {X 0,Y 96.524,Z 342.9,A -85,B 0,C 180,E1 -26817.391,E2 -26817.391} C_VEL
LIN {X 0,Y 95.981,Z 341.765,A -85,B 0,C 180,E1 -26819.999,E2 -26819.999} C_VEL
LIN {X 0,Y 95.183,Z 341.664,A -85,B 0,C 180,E1 -26829.562,E2 -26829.562} C_VEL
LIN {X 0,Y 99.049,Z 345.002,A -85,B 0,C 180,E1 -26844.992,E2 -26844.992} C_VEL
LIN {X 0,Y 100.235,Z 347.714,A -85,B 0,C 180,E1 -26847.678,E2 -26847.678} C_VEL
LIN {X 0,Y 103.421,Z 350.731,A -85,B 0,C 180,E1 -26852.65,E2 -26852.65} C_VEL
LIN {X 0,Y 105.595,Z 354.066,A -85,B 0,C 180,E1 -26855.616,E2 -26855.616} C_VEL
LIN {X 0,Y 107.208,Z 355.793,A -85,B 0,C 180,E1 -26857.489,E2 -26857.489} C_VEL
LIN {X 0,Y 109.823,Z 359.441,A -85,B 0,C 180,E1 -26860.312,E2 -26860.312} C_VEL
LIN {X 0,Y 114.917,Z 367.102,A -85,B 0,C 180,E1 -26864.998,E2 -26864.998} C_VEL
LIN {X 0,Y 119.987,Z 375.895,A -85,B 0,C 180,E1 -26868.963,E2 -26868.963} C_VEL
LIN {X 0,Y 124.715,Z 385.546,A -85,B 0,C 180,E1 -26872.249,E2 -26872.249} C_VEL
LIN {X 0,Y 126.626,Z 390.338,A -85,B 0,C 180,E1 -26873.528,E2 -26873.528} C_VEL
LIN {X 0,Y 123.058,Z 432.555,A -85,B 0,C 180,E1 -26875.454,E2 -26875.454} C_VEL
LIN {X 0,Y 120.988,Z 446.004,A -85,B 0,C 180,E1 -26876.622,E2 -26876.622} C_VEL
LIN {X 0,Y 118.294,Z 458.894,A -85,B 0,C 180,E1 -26878.423,E2 -26878.423} C_VEL
LIN {X 0,Y 114.821,Z 470.726,A -85,B 0,C 180,E1 -26880.676,E2 -26880.676} C_VEL
LIN {X 0,Y 110.957,Z 482.072,A -85,B 0,C 180,E1 -26883.675,E2 -26883.675} C_VEL
LIN {X 0,Y 107.285,Z 491.271,A -85,B 0,C 180,E1 -26886.85,E2 -26886.85} C_VEL
LIN {X 0,Y 103.2,Z 500.7,A -85,B 0,C 180,E1 -26891.121,E2 -26891.121} C_VEL
LIN {X 0,Y 98.884,Z 509.824,A -85,B 0,C 180,E1 -26896.639,E2 -26896.639} C_VEL
LIN {X 0,Y 95.527,Z 517.167,A -85,B 0,C 180,E1 -26902.596,E2 -26902.596} C_VEL
LIN {X 0,Y 93.478,Z 522.123,A -85,B 0,C 180,E1 -26907.839,E2 -26907.839} C_VEL
LIN {X 0,Y 91.681,Z 527.212,A -85,B 0,C 180,E1 -26914.773,E2 -26914.773} C_VEL
LIN {X 0,Y 90.75,Z 530.683,A -85,B 0,C 180,E1 -26921.157,E2 -26921.157} C_VEL
LIN {X 0,Y 90.776,Z 533.363,A -85,B 0,C 180,E1 -26928.033,E2 -26928.033} C_VEL
LIN {X 0,Y 91.327,Z 534.625,A -85,B 0,C 180,E1 -26932.622,E2 -26932.622} C_VEL
LIN {X 0,Y 92.33,Z 535.42,A -85,B 0,C 180,E1 -26937.167,E2 -26937.167} C_VEL
LIN {X 0,Y 93.829,Z 535.808,A -85,B 0,C 180,E1 -26941.614,E2 -26941.614} C_VEL
LIN {X 0,Y 96.137,Z 535.761,A -85,B 0,C 180,E1 -26946.473,E2 -26946.473} C_VEL
LIN {X 0,Y 101.214,Z 534.416,A -85,B 0,C 180,E1 -26953.968,E2 -26953.968} C_VEL
LIN {X 0,Y 104.851,Z 532.981,A -85,B 0,C 180,E1 -26957.912,E2 -26957.912} C_VEL
LIN {X 0,Y 110.331,Z 530.215,A -85,B 0,C 180,E1 -26962.763,E2 -26962.763} C_VEL
LIN {X 0,Y 116.868,Z 526.227,A -85,B 0,C 180,E1 -26967.332,E2 -26967.332} C_VEL
LIN {X 0,Y 124.058,Z 521,A -85,B 0,C 180,E1 -26971.402,E2 -26971.402} C_VEL
LIN {X 0,Y 131.768,Z 514.303,A -85,B 0,C 180,E1 -26975.043,E2 -26975.043} C_VEL
LIN {X 0,Y 139.968,Z 505.894,A -85,B 0,C 180,E1 -26978.253,E2 -26978.253} C_VEL
LIN {X 0,Y 147.811,Z 496.286,A -85,B 0,C 180,E1 -26980.839,E2 -26980.839} C_VEL
LIN {X 0,Y 154.472,Z 486.376,A -85,B 0,C 180,E1 -26982.815,E2 -26982.815} C_VEL
LIN {X 0,Y 160.502,Z 475.531,A -85,B 0,C 180,E1 -26984.418,E2 -26984.418} C_VEL
LIN {X 0,Y 165.237,Z 464.9,A -85,B 0,C 180,E1 -26985.635,E2 -26985.635} C_VEL
LIN {X 0,Y 169.153,Z 453.842,A -85,B 0,C 180,E1 -26986.538,E2 -26986.538} C_VEL
LIN {X 0,Y 172.31,Z 441.477,A -85,B 0,C 180,E1 -26987.288,E2 -26987.288} C_VEL
LIN {X 0,Y 174.299,Z 429.451,A -85,B 0,C 180,E1 -26987.781,E2 -26987.781} C_VEL
LIN {X 0,Y 171.424,Z 423.044,A -85,B 0,C 180,E1 -26991.584,E2 -26991.584} C_VEL
LIN {X 0,Y 169.338,Z 418.648,A -85,B 0,C 180,E1 -26995.109,E2 -26995.109} C_VEL
LIN {X 0,Y 168.006,Z 415.789,A -85,B 0,C 180,E1 -26998.107,E2 -26998.107} C_VEL
LIN {X 0,Y 166.675,Z 412.515,A -85,B 0,C 180,E1 -27003.022,E2 -27003.022} C_VEL
LIN {X 0,Y 166.395,Z 412.122,A -85,B 0,C 180,E1 -27004.846,E2 -27004.846} C_VEL
LIN {X 0,Y 166.552,Z 412.319,A -85,B 0,C 180,E1 -27010.791,E2 -27010.791} C_VEL
LIN {X 0,Y 167.801,Z 415.872,A -85,B 0,C 180,E1 -27016.022,E2 -27016.022} C_VEL
LIN {X 0,Y 168.378,Z 416.898,A -85,B 0,C 180,E1 -27017.438,E2 -27017.438} C_VEL
LIN {X 0,Y 169.758,Z 420.71,A -85,B 0,C 180,E1 -27020.446,E2 -27020.446} C_VEL
LIN {X 0,Y 171.107,Z 424.548,A -85,B 0,C 180,E1 -27022.808,E2 -27022.808} C_VEL
LIN {X 0,Y 172.984,Z 430.267,A -85,B 0,C 180,E1 -27025.574,E2 -27025.574} C_VEL
LIN {X 0,Y 173.949,Z 433.447,A -85,B 0,C 180,E1 -27026.907,E2 -27026.907} C_VEL
LIN {X 0,Y 171.851,Z 446.084,A -85,B 0,C 180,E1 -27027.391,E2 -27027.391} C_VEL
LIN {X 0,Y 168.557,Z 458.583,A -85,B 0,C 180,E1 -27028.059,E2 -27028.059} C_VEL
LIN {X 0,Y 163.784,Z 471.438,A -85,B 0,C 180,E1 -27029.047,E2 -27029.047} C_VEL
LIN {X 0,Y 157.744,Z 483.828,A -85,B 0,C 180,E1 -27030.329,E2 -27030.329} C_VEL
LIN {X 0,Y 151.187,Z 494.688,A -85,B 0,C 180,E1 -27031.975,E2 -27031.975} C_VEL
LIN {X 0,Y 144.092,Z 504.444,A -85,B 0,C 180,E1 -27033.996,E2 -27033.996} C_VEL
LIN {X 0,Y 135.866,Z 513.929,A -85,B 0,C 180,E1 -27036.708,E2 -27036.708} C_VEL
LIN {X 0,Y 128.075,Z 521.502,A -85,B 0,C 180,E1 -27039.812,E2 -27039.812} C_VEL
LIN {X 0,Y 120.654,Z 527.628,A -85,B 0,C 180,E1 -27043.28,E2 -27043.28} C_VEL
LIN {X 0,Y 113.904,Z 532.514,A -85,B 0,C 180,E1 -27047.265,E2 -27047.265} C_VEL
LIN {X 0,Y 107.914,Z 536.311,A -85,B 0,C 180,E1 -27051.787,E2 -27051.787} C_VEL
LIN {X 0,Y 102.568,Z 539.124,A -85,B 0,C 180,E1 -27056.766,E2 -27056.766} C_VEL
LIN {X 0,Y 96.824,Z 541.445,A -85,B 0,C 180,E1 -27064.189,E2 -27064.189} C_VEL
LIN {X 0,Y 94.65,Z 542.037,A -85,B 0,C 180,E1 -27068.214,E2 -27068.214} C_VEL
LIN {X 0,Y 91.928,Z 542.017,A -85,B 0,C 180,E1 -27076.748,E2 -27076.748} C_VEL
LIN {X 0,Y 91.079,Z 540.481,A -85,B 0,C 180,E1 -27085.581,E2 -27085.581} C_VEL
LIN {X 0,Y 91.177,Z 539.093,A -85,B 0,C 180,E1 -27090.007,E2 -27090.007} C_VEL
LIN {X 0,Y 91.118,Z 536.124,A -85,B 0,C 180,E1 -27096.65,E2 -27096.65} C_VEL
LIN {X 0,Y 91.857,Z 532.063,A -85,B 0,C 180,E1 -27103.276,E2 -27103.276} C_VEL
LIN {X 0,Y 93.919,Z 525.77,A -85,B 0,C 180,E1 -27110.827,E2 -27110.827} C_VEL
LIN {X 0,Y 96.974,Z 518.912,A -85,B 0,C 180,E1 -27116.94,E2 -27116.94} C_VEL
LIN {X 0,Y 100.56,Z 510.76,A -85,B 0,C 180,E1 -27122.471,E2 -27122.471} C_VEL
LIN {X 0,Y 104.938,Z 501.478,A -85,B 0,C 180,E1 -27127.074,E2 -27127.074} C_VEL
LIN {X 0,Y 109.407,Z 490.536,A -85,B 0,C 180,E1 -27131.187,E2 -27131.187} C_VEL
LIN {X 0,Y 109.465,Z 490.38,A -85,B 0,C 180,E1 -27131.237,E2 -27131.237} C_VEL
LIN {X 0,Y 110.717,Z 485.54,A -85,B 0,C 180,E1 -27132.888,E2 -27132.888} C_VEL
LIN {X 0,Y 111.402,Z 477.396,A -85,B 0,C 180,E1 -27135.791,E2 -27135.791} C_VEL
LIN {X 0,Y 111.986,Z 468.883,A -85,B 0,C 180,E1 -27138.365,E2 -27138.365} C_VEL
LIN {X 0,Y 112.995,Z 463.47,A -85,B 0,C 180,E1 -27139.449,E2 -27139.449} C_VEL
LIN {X 0,Y 115.99,Z 450.325,A -85,B 0,C 180,E1 -27141.105,E2 -27141.105} C_VEL
LIN {X 0,Y 118.014,Z 437.085,A -85,B 0,C 180,E1 -27142.168,E2 -27142.168} C_VEL
LIN {X 0,Y 120.946,Z 400.258,A -85,B 0,C 180,E1 -27143.967,E2 -27143.967} C_VEL
LIN {X 0,Y 120.682,Z 394.864,A -85,B 0,C 180,E1 -27144.572,E2 -27144.572} C_VEL
LIN {X 0,Y 117.417,Z 384.294,A -85,B 0,C 180,E1 -27147.329,E2 -27147.329} C_VEL
LIN {X 0,Y 115.206,Z 378.903,A -85,B 0,C 180,E1 -27149.206,E2 -27149.206} C_VEL
LIN {X 0,Y 111.116,Z 371.593,A -85,B 0,C 180,E1 -27152.822,E2 -27152.822} C_VEL
LIN {X 0,Y 107.038,Z 365.133,A -85,B 0,C 180,E1 -27157.008,E2 -27157.008} C_VEL
LIN {X 0,Y 104.305,Z 361.072,A -85,B 0,C 180,E1 -27160.311,E2 -27160.311} C_VEL
LIN {X 0,Y 101.857,Z 357.694,A -85,B 0,C 180,E1 -27163.72,E2 -27163.72} C_VEL
LIN {X 0,Y 101.109,Z 356.633,A -85,B 0,C 180,E1 -27164.89,E2 -27164.89} C_VEL
LIN {X 0,Y 98.772,Z 354.001,A -85,B 0,C 180,E1 -27168.975,E2 -27168.975} C_VEL
LIN {X 0,Y 97.641,Z 351.481,A -85,B 0,C 180,E1 -27171.722,E2 -27171.722} C_VEL
LIN {X 0,Y 95.306,Z 349.59,A -85,B 0,C 180,E1 -27178.679,E2 -27178.679} C_VEL
LIN {X 0,Y 94.873,Z 348.766,A -85,B 0,C 180,E1 -27181.06,E2 -27181.06} C_VEL
LIN {X 0,Y 94.301,Z 348.751,A -85,B 0,C 180,E1 -27189.634,E2 -27189.634} C_VEL
LIN {X 0,Y 97.515,Z 351.811,A -85,B 0,C 180,E1 -27203.719,E2 -27203.719} C_VEL
LIN {X 0,Y 98.993,Z 354.807,A -85,B 0,C 180,E1 -27207.195,E2 -27207.195} C_VEL
LIN {X 0,Y 101.399,Z 357.083,A -85,B 0,C 180,E1 -27211.196,E2 -27211.196} C_VEL
LIN {X 0,Y 103.714,Z 360.63,A -85,B 0,C 180,E1 -27214.576,E2 -27214.576} C_VEL
LIN {X 0,Y 104.967,Z 362.198,A -85,B 0,C 180,E1 -27216.159,E2 -27216.159} C_VEL
LIN {X 0,Y 108.02,Z 366.826,A -85,B 0,C 180,E1 -27219.695,E2 -27219.695} C_VEL
LIN {X 0,Y 111.924,Z 372.898,A -85,B 0,C 180,E1 -27223.529,E2 -27223.529} C_VEL
LIN {X 0,Y 116.308,Z 380.882,A -85,B 0,C 180,E1 -27227.287,E2 -27227.287} C_VEL
LIN {X 0,Y 120.702,Z 390.346,A -85,B 0,C 180,E1 -27230.651,E2 -27230.651} C_VEL
LIN {X 0,Y 121.479,Z 392.222,A -85,B 0,C 180,E1 -27231.217,E2 -27231.217} C_VEL
LIN {X 0,Y 117.931,Z 432.941,A -85,B 0,C 180,E1 -27233.126,E2 -27233.126} C_VEL
LIN {X 0,Y 115.798,Z 446.169,A -85,B 0,C 180,E1 -27234.284,E2 -27234.284} C_VEL
LIN {X 0,Y 113.123,Z 458.427,A -85,B 0,C 180,E1 -27235.998,E2 -27235.998} C_VEL
LIN {X 0,Y 109.782,Z 469.618,A -85,B 0,C 180,E1 -27238.114,E2 -27238.114} C_VEL
LIN {X 0,Y 106.077,Z 479.942,A -85,B 0,C 180,E1 -27240.744,E2 -27240.744} C_VEL
LIN {X 0,Y 102.699,Z 488.446,A -85,B 0,C 180,E1 -27243.582,E2 -27243.582} C_VEL
LIN {X 0,Y 98.151,Z 498.434,A -85,B 0,C 180,E1 -27247.911,E2 -27247.911} C_VEL
LIN {X 0,Y 94.118,Z 506.627,A -85,B 0,C 180,E1 -27252.615,E2 -27252.615} C_VEL
LIN {X 0,Y 90.083,Z 514.667,A -85,B 0,C 180,E1 -27258.746,E2 -27258.746} C_VEL
LIN {X 0,Y 87.091,Z 521.073,A -85,B 0,C 180,E1 -27265.365,E2 -27265.365} C_VEL
LIN {X 0,Y 85.075,Z 526.088,A -85,B 0,C 180,E1 -27272.214,E2 -27272.214} C_VEL
LIN {X 0,Y 83.795,Z 530.159,A -85,B 0,C 180,E1 -27279.649,E2 -27279.649} C_VEL
LIN {X 0,Y 83.51,Z 532.22,A -85,B 0,C 180,E1 -27284.616,E2 -27284.616} C_VEL
LIN {X 0,Y 84.382,Z 534.849,A -85,B 0,C 180,E1 -27293.63,E2 -27293.63} C_VEL
LIN {X 0,Y 85.786,Z 535.768,A -85,B 0,C 180,E1 -27299.434,E2 -27299.434} C_VEL
LIN {X 0,Y 89.744,Z 536.046,A -85,B 0,C 180,E1 -27308.455,E2 -27308.455} C_VEL
LIN {X 0,Y 92.692,Z 535.482,A -85,B 0,C 180,E1 -27313.021,E2 -27313.021} C_VEL
LIN {X 0,Y 99.266,Z 533.312,A -85,B 0,C 180,E1 -27320.418,E2 -27320.418} C_VEL
LIN {X 0,Y 105.982,Z 530.166,A -85,B 0,C 180,E1 -27325.977,E2 -27325.977} C_VEL
LIN {X 0,Y 113.024,Z 526.057,A -85,B 0,C 180,E1 -27330.509,E2 -27330.509} C_VEL
LIN {X 0,Y 122.002,Z 519.636,A -85,B 0,C 180,E1 -27335.12,E2 -27335.12} C_VEL
LIN {X 0,Y 130.199,Z 512.564,A -85,B 0,C 180,E1 -27338.599,E2 -27338.599} C_VEL
LIN {X 0,Y 137.406,Z 505.276,A -85,B 0,C 180,E1 -27341.11,E2 -27341.11} C_VEL
LIN {X 0,Y 145.303,Z 495.712,A -85,B 0,C 180,E1 -27343.531,E2 -27343.531} C_VEL
LIN {X 0,Y 152.45,Z 485.245,A -85,B 0,C 180,E1 -27345.473,E2 -27345.473} C_VEL
LIN {X 0,Y 158.671,Z 474.016,A -85,B 0,C 180,E1 -27347,E2 -27347} C_VEL
LIN {X 0,Y 164.132,Z 461.33,A -85,B 0,C 180,E1 -27348.284,E2 -27348.284} C_VEL
LIN {X 0,Y 167.998,Z 449.585,A -85,B 0,C 180,E1 -27349.099,E2 -27349.099} C_VEL
LIN {X 0,Y 170.956,Z 436.576,A -85,B 0,C 180,E1 -27349.722,E2 -27349.722} C_VEL
LIN {X 0,Y 171.418,Z 433.533,A -85,B 0,C 180,E1 -27349.887,E2 -27349.887} C_VEL
LIN {X 0,Y 169.165,Z 427.89,A -85,B 0,C 180,E1 -27353.627,E2 -27353.627} C_VEL
LIN {X 0,Y 167.773,Z 424.73,A -85,B 0,C 180,E1 -27356.398,E2 -27356.398} C_VEL
LIN {X 0,Y 166.831,Z 422.543,A -85,B 0,C 180,E1 -27358.794,E2 -27358.794} C_VEL
LIN {X 0,Y 165.691,Z 419.307,A -85,B 0,C 180,E1 -27363.648,E2 -27363.648} C_VEL
LIN {X 0,Y 165.52,Z 419.236,A -85,B 0,C 180,E1 -27369.779,E2 -27369.779} C_VEL
LIN {X 0,Y 165.673,Z 419.876,A -85,B 0,C 180,E1 -27371.142,E2 -27371.142} C_VEL
LIN {X 0,Y 167.177,Z 423.614,A -85,B 0,C 180,E1 -27376.766,E2 -27376.766} C_VEL
LIN {X 0,Y 168.308,Z 427.097,A -85,B 0,C 180,E1 -27379.516,E2 -27379.516} C_VEL
LIN {X 0,Y 169.64,Z 431.358,A -85,B 0,C 180,E1 -27382.133,E2 -27382.133} C_VEL
LIN {X 0,Y 171.144,Z 436.893,A -85,B 0,C 180,E1 -27384.773,E2 -27384.773} C_VEL
LIN {X 0,Y 168.638,Z 449.399,A -85,B 0,C 180,E1 -27385.287,E2 -27385.287} C_VEL
LIN {X 0,Y 165.001,Z 461.545,A -85,B 0,C 180,E1 -27385.966,E2 -27385.966} C_VEL
LIN {X 0,Y 160.493,Z 472.869,A -85,B 0,C 180,E1 -27386.856,E2 -27386.856} C_VEL
LIN {X 0,Y 155.075,Z 483.519,A -85,B 0,C 180,E1 -27387.913,E2 -27387.913} C_VEL
LIN {X 0,Y 149.066,Z 493.324,A -85,B 0,C 180,E1 -27389.292,E2 -27389.292} C_VEL
LIN {X 0,Y 143.123,Z 501.472,A -85,B 0,C 180,E1 -27390.768,E2 -27390.768} C_VEL
LIN {X 0,Y 136.002,Z 509.954,A -85,B 0,C 180,E1 -27392.897,E2 -27392.897} C_VEL
LIN {X 0,Y 127.687,Z 518.244,A -85,B 0,C 180,E1 -27395.732,E2 -27395.732} C_VEL
LIN {X 0,Y 119.732,Z 524.954,A -85,B 0,C 180,E1 -27398.954,E2 -27398.954} C_VEL
LIN {X 0,Y 111.061,Z 531.15,A -85,B 0,C 180,E1 -27403.313,E2 -27403.313} C_VEL
LIN {X 0,Y 104.053,Z 535.416,A -85,B 0,C 180,E1 -27407.986,E2 -27407.986} C_VEL
LIN {X 0,Y 100.461,Z 537.334,A -85,B 0,C 180,E1 -27410.986,E2 -27410.986} C_VEL
LIN {X 0,Y 93.387,Z 540.346,A -85,B 0,C 180,E1 -27418.219,E2 -27418.219} C_VEL
LIN {X 0,Y 90.483,Z 541.277,A -85,B 0,C 180,E1 -27422.231,E2 -27422.231} C_VEL
LIN {X 0,Y 88.065,Z 541.802,A -85,B 0,C 180,E1 -27426.491,E2 -27426.491} C_VEL
LIN {X 0,Y 85.006,Z 541.692,A -85,B 0,C 180,E1 -27435.647,E2 -27435.647} C_VEL
LIN {X 0,Y 84.019,Z 540.074,A -85,B 0,C 180,E1 -27445.209,E2 -27445.209} C_VEL
LIN {X 0,Y 84.089,Z 538.615,A -85,B 0,C 180,E1 -27450.007,E2 -27450.007} C_VEL
LIN {X 0,Y 84.074,Z 535.565,A -85,B 0,C 180,E1 -27457.21,E2 -27457.21} C_VEL
LIN {X 0,Y 84.933,Z 531.412,A -85,B 0,C 180,E1 -27464.381,E2 -27464.381} C_VEL
LIN {X 0,Y 87.293,Z 525.02,A -85,B 0,C 180,E1 -27472.491,E2 -27472.491} C_VEL
LIN {X 0,Y 90.634,Z 518.048,A -85,B 0,C 180,E1 -27478.996,E2 -27478.996} C_VEL
LIN {X 0,Y 93.857,Z 511.283,A -85,B 0,C 180,E1 -27483.828,E2 -27483.828} C_VEL
LIN {X 0,Y 97.513,Z 504.095,A -85,B 0,C 180,E1 -27487.784,E2 -27487.784} C_VEL
LIN {X 0,Y 102.145,Z 493.891,A -85,B 0,C 180,E1 -27492.139,E2 -27492.139} C_VEL
LIN {X 0,Y 105.708,Z 485.157,A -85,B 0,C 180,E1 -27494.95,E2 -27494.95} C_VEL
LIN {X 0,Y 109.644,Z 474.527,A -85,B 0,C 180,E1 -27497.495,E2 -27497.495} C_VEL
LIN {X 0,Y 112.995,Z 463.47,A -85,B 0,C 180,E1 -27499.449,E2 -27499.449} C_VEL
LIN {X 0,Y 113.901,Z 458.011,A -85,B 0,C 180,E1 -27500.434,E2 -27500.434} C_VEL
LIN {X 0,Y 113.809,Z 448.9,A -85,B 0,C 180,E1 -27502.451,E2 -27502.451} C_VEL
LIN {X 0,Y 113.268,Z 439.664,A -85,B 0,C 180,E1 -27504.262,E2 -27504.262} C_VEL
LIN {X 0,Y 113.421,Z 433.882,A -85,B 0,C 180,E1 -27504.887,E2 -27504.887} C_VEL
LIN {X 0,Y 116.166,Z 400.758,A -85,B 0,C 180,E1 -27506.491,E2 -27506.491} C_VEL
LIN {X 0,Y 115.965,Z 397.208,A -85,B 0,C 180,E1 -27506.944,E2 -27506.944} C_VEL
LIN {X 0,Y 112.882,Z 386.919,A -85,B 0,C 180,E1 -27509.896,E2 -27509.896} C_VEL
LIN {X 0,Y 111.082,Z 382.633,A -85,B 0,C 180,E1 -27511.605,E2 -27511.605} C_VEL
LIN {X 0,Y 106.782,Z 374.763,A -85,B 0,C 180,E1 -27515.975,E2 -27515.975} C_VEL
LIN {X 0,Y 103.494,Z 369.609,A -85,B 0,C 180,E1 -27519.892,E2 -27519.892} C_VEL
LIN {X 0,Y 101.798,Z 366.96,A -85,B 0,C 180,E1 -27522.227,E2 -27522.227} C_VEL
LIN {X 0,Y 99.384,Z 363.27,A -85,B 0,C 180,E1 -27526.054,E2 -27526.054} C_VEL
LIN {X 0,Y 97.035,Z 360.271,A -85,B 0,C 180,E1 -27530.637,E2 -27530.637} C_VEL
LIN {X 0,Y 96.303,Z 358.39,A -85,B 0,C 180,E1 -27532.662,E2 -27532.662} C_VEL
LIN {X 0,Y 94.05,Z 356.085,A -85,B 0,C 180,E1 -27540.534,E2 -27540.534} C_VEL
LIN {X 0,Y 93.548,Z 355.622,A -85,B 0,C 180,E1 -27544.308,E2 -27544.308} C_VEL
LIN {X 0,Y 93.465,Z 355.98,A -85,B 0,C 180,E1 -27550.798,E2 -27550.798} C_VEL
LIN {X 0,Y 96.122,Z 358.791,A -85,B 0,C 180,E1 -27562.655,E2 -27562.655} C_VEL
LIN {X 0,Y 97.766,Z 361.867,A -85,B 0,C 180,E1 -27566.697,E2 -27566.697} C_VEL
LIN {X 0,Y 99.552,Z 363.711,A -85,B 0,C 180,E1 -27569.89,E2 -27569.89} C_VEL
LIN {X 0,Y 102.204,Z 367.588,A -85,B 0,C 180,E1 -27573.966,E2 -27573.966} C_VEL
LIN {X 0,Y 105.47,Z 372.862,A -85,B 0,C 180,E1 -27578.17,E2 -27578.17} C_VEL
LIN {X 0,Y 108.585,Z 377.922,A -85,B 0,C 180,E1 -27581.549,E2 -27581.549} C_VEL
LIN {X 0,Y 112.83,Z 386.073,A -85,B 0,C 180,E1 -27585.587,E2 -27585.587} C_VEL
LIN {X 0,Y 116.589,Z 394.617,A -85,B 0,C 180,E1 -27588.78,E2 -27588.78} C_VEL
LIN {X 0,Y 113.005,Z 433.417,A -85,B 0,C 180,E1 -27590.597,E2 -27590.597} C_VEL
LIN {X 0,Y 110.743,Z 446.691,A -85,B 0,C 180,E1 -27591.768,E2 -27591.768} C_VEL
LIN {X 0,Y 107.889,Z 459.001,A -85,B 0,C 180,E1 -27593.523,E2 -27593.523} C_VEL
LIN {X 0,Y 104.367,Z 470.114,A -85,B 0,C 180,E1 -27595.663,E2 -27595.663} C_VEL
LIN {X 0,Y 100.459,Z 480.395,A -85,B 0,C 180,E1 -27598.346,E2 -27598.346} C_VEL
LIN {X 0,Y 96.535,Z 489.477,A -85,B 0,C 180,E1 -27601.486,E2 -27601.486} C_VEL
LIN {X 0,Y 91.656,Z 499.551,A -85,B 0,C 180,E1 -27606.135,E2 -27606.135} C_VEL
LIN {X 0,Y 87.313,Z 507.753,A -85,B 0,C 180,E1 -27611.211,E2 -27611.211} C_VEL
LIN {X 0,Y 83.047,Z 515.596,A -85,B 0,C 180,E1 -27617.779,E2 -27617.779} C_VEL
LIN {X 0,Y 79.943,Z 521.864,A -85,B 0,C 180,E1 -27624.949,E2 -27624.949} C_VEL
LIN {X 0,Y 77.938,Z 526.562,A -85,B 0,C 180,E1 -27632.046,E2 -27632.046} C_VEL
LIN {X 0,Y 76.605,Z 530.744,A -85,B 0,C 180,E1 -27640.565,E2 -27640.565} C_VEL
LIN {X 0,Y 76.424,Z 532.759,A -85,B 0,C 180,E1 -27646.006,E2 -27646.006} C_VEL
LIN {X 0,Y 77.434,Z 535.072,A -85,B 0,C 180,E1 -27654.825,E2 -27654.825} C_VEL
LIN {X 0,Y 79.4,Z 536.116,A -85,B 0,C 180,E1 -27662.069,E2 -27662.069} C_VEL
LIN {X 0,Y 83.509,Z 536.325,A -85,B 0,C 180,E1 -27670.764,E2 -27670.764} C_VEL
LIN {X 0,Y 87.376,Z 535.638,A -85,B 0,C 180,E1 -27676.367,E2 -27676.367} C_VEL
LIN {X 0,Y 93.858,Z 533.652,A -85,B 0,C 180,E1 -27683.2,E2 -27683.2} C_VEL
LIN {X 0,Y 101.997,Z 530.077,A -85,B 0,C 180,E1 -27689.45,E2 -27689.45} C_VEL
LIN {X 0,Y 109.542,Z 525.848,A -85,B 0,C 180,E1 -27693.91,E2 -27693.91} C_VEL
LIN {X 0,Y 117.66,Z 520.345,A -85,B 0,C 180,E1 -27697.78,E2 -27697.78} C_VEL
LIN {X 0,Y 126.205,Z 513.372,A -85,B 0,C 180,E1 -27701.189,E2 -27701.189} C_VEL
LIN {X 0,Y 133.667,Z 506.201,A -85,B 0,C 180,E1 -27703.631,E2 -27703.631} C_VEL
LIN {X 0,Y 141.557,Z 497.187,A -85,B 0,C 180,E1 -27705.886,E2 -27705.886} C_VEL
LIN {X 0,Y 149.176,Z 486.55,A -85,B 0,C 180,E1 -27707.822,E2 -27707.822} C_VEL
LIN {X 0,Y 155.563,Z 475.625,A -85,B 0,C 180,E1 -27709.277,E2 -27709.277} C_VEL
LIN {X 0,Y 160.954,Z 463.875,A -85,B 0,C 180,E1 -27710.47,E2 -27710.47} C_VEL
LIN {X 0,Y 165.341,Z 451.433,A -85,B 0,C 180,E1 -27711.317,E2 -27711.317} C_VEL
LIN {X 0,Y 168.583,Z 438.327,A -85,B 0,C 180,E1 -27711.956,E2 -27711.956} C_VEL
LIN {X 0,Y 168.617,Z 437.6,A -85,B 0,C 180,E1 -27712.102,E2 -27712.102} C_VEL
LIN {X 0,Y 167.008,Z 432.702,A -85,B 0,C 180,E1 -27715.777,E2 -27715.777} C_VEL
LIN {X 0,Y 165.693,Z 429.324,A -85,B 0,C 180,E1 -27719.393,E2 -27719.393} C_VEL
LIN {X 0,Y 164.706,Z 426.269,A -85,B 0,C 180,E1 -27724.283,E2 -27724.283} C_VEL
LIN {X 0,Y 164.642,Z 426.304,A -85,B 0,C 180,E1 -27729.832,E2 -27729.832} C_VEL
LIN {X 0,Y 166.033,Z 430.452,A -85,B 0,C 180,E1 -27736.207,E2 -27736.207} C_VEL
LIN {X 0,Y 167.139,Z 434.586,A -85,B 0,C 180,E1 -27739.338,E2 -27739.338} C_VEL
LIN {X 0,Y 168.335,Z 439.979,A -85,B 0,C 180,E1 -27742.378,E2 -27742.378} C_VEL
LIN {X 0,Y 168.435,Z 440.514,A -85,B 0,C 180,E1 -27742.625,E2 -27742.625} C_VEL
LIN {X 0,Y 165.777,Z 452.038,A -85,B 0,C 180,E1 -27743.105,E2 -27743.105} C_VEL
LIN {X 0,Y 161.796,Z 464.101,A -85,B 0,C 180,E1 -27743.787,E2 -27743.787} C_VEL
LIN {X 0,Y 156.639,Z 475.827,A -85,B 0,C 180,E1 -27744.702,E2 -27744.702} C_VEL
LIN {X 0,Y 150.338,Z 487.108,A -85,B 0,C 180,E1 -27745.866,E2 -27745.866} C_VEL
LIN {X 0,Y 143.44,Z 497.282,A -85,B 0,C 180,E1 -27747.381,E2 -27747.381} C_VEL
LIN {X 0,Y 136.684,Z 505.63,A -85,B 0,C 180,E1 -27749.071,E2 -27749.071} C_VEL
LIN {X 0,Y 127.915,Z 514.712,A -85,B 0,C 180,E1 -27751.623,E2 -27751.623} C_VEL
LIN {X 0,Y 119.498,Z 522.055,A -85,B 0,C 180,E1 -27754.585,E2 -27754.585} C_VEL
LIN {X 0,Y 111.406,Z 527.977,A -85,B 0,C 180,E1 -27757.959,E2 -27757.959} C_VEL
LIN {X 0,Y 103.899,Z 532.677,A -85,B 0,C 180,E1 -27761.93,E2 -27761.93} C_VEL
LIN {X 0,Y 98.247,Z 535.717,A -85,B 0,C 180,E1 -27765.672,E2 -27765.672} C_VEL
LIN {X 0,Y 91.006,Z 538.946,A -85,B 0,C 180,E1 -27771.853,E2 -27771.853} C_VEL
LIN {X 0,Y 84.24,Z 541.094,A -85,B 0,C 180,E1 -27779.971,E2 -27779.971} C_VEL
LIN {X 0,Y 79.574,Z 541.648,A -85,B 0,C 180,E1 -27789.32,E2 -27789.32} C_VEL
LIN {X 0,Y 77.25,Z 540.714,A -85,B 0,C 180,E1 -27799.524,E2 -27799.524} C_VEL
LIN {X 0,Y 76.952,Z 539.638,A -85,B 0,C 180,E1 -27804.768,E2 -27804.768} C_VEL
LIN {X 0,Y 76.993,Z 538.133,A -85,B 0,C 180,E1 -27810.008,E2 -27810.008} C_VEL
LIN {X 0,Y 77.015,Z 534.996,A -85,B 0,C 180,E1 -27817.875,E2 -27817.875} C_VEL
LIN {X 0,Y 78.026,Z 530.75,A -85,B 0,C 180,E1 -27825.685,E2 -27825.685} C_VEL
LIN {X 0,Y 80.752,Z 524.262,A -85,B 0,C 180,E1 -27834.427,E2 -27834.427} C_VEL
LIN {X 0,Y 84.41,Z 517.137,A -85,B 0,C 180,E1 -27841.365,E2 -27841.365} C_VEL
LIN {X 0,Y 87.73,Z 510.709,A -85,B 0,C 180,E1 -27846.151,E2 -27846.151} C_VEL
LIN {X 0,Y 91.972,Z 502.952,A -85,B 0,C 180,E1 -27850.514,E2 -27850.514} C_VEL
LIN {X 0,Y 96.43,Z 493.662,A -85,B 0,C 180,E1 -27854.554,E2 -27854.554} C_VEL
LIN {X 0,Y 100.205,Z 484.932,A -85,B 0,C 180,E1 -27857.436,E2 -27857.436} C_VEL
LIN {X 0,Y 104.344,Z 474.314,A -85,B 0,C 180,E1 -27860.018,E2 -27860.018} C_VEL
LIN {X 0,Y 108.029,Z 462.633,A -85,B 0,C 180,E1 -27862.082,E2 -27862.082} C_VEL
LIN {X 0,Y 111.149,Z 449.374,A -85,B 0,C 180,E1 -27863.733,E2 -27863.733} C_VEL
LIN {X 0,Y 113.145,Z 436.721,A -85,B 0,C 180,E1 -27864.724,E2 -27864.724} C_VEL
LIN {X 0,Y 113.421,Z 433.882,A -85,B 0,C 180,E1 -27864.887,E2 -27864.887} C_VEL
LIN {X 0,Y 113.504,Z 428.074,A -85,B 0,C 180,E1 -27865.459,E2 -27865.459} C_VEL
LIN {X 0,Y 111.402,Z 409.286,A -85,B 0,C 180,E1 -27868.555,E2 -27868.555} C_VEL
LIN {X 0,Y 111.498,Z 403.462,A -85,B 0,C 180,E1 -27869.083,E2 -27869.083} C_VEL
LIN {X 0,Y 111.515,Z 399.737,A -85,B 0,C 180,E1 -27869.461,E2 -27869.461} C_VEL
LIN {X 0,Y 108.78,Z 390.126,A -85,B 0,C 180,E1 -27872.46,E2 -27872.46} C_VEL
LIN {X 0,Y 105.921,Z 384.051,A -85,B 0,C 180,E1 -27875.534,E2 -27875.534} C_VEL
LIN {X 0,Y 102.282,Z 377.314,A -85,B 0,C 180,E1 -27880.031,E2 -27880.031} C_VEL
LIN {X 0,Y 99.79,Z 373.271,A -85,B 0,C 180,E1 -27883.637,E2 -27883.637} C_VEL
LIN {X 0,Y 97.561,Z 369.741,A -85,B 0,C 180,E1 -27887.518,E2 -27887.518} C_VEL
LIN {X 0,Y 95.399,Z 366.54,A -85,B 0,C 180,E1 -27892.326,E2 -27892.326} C_VEL
LIN {X 0,Y 94.811,Z 365.092,A -85,B 0,C 180,E1 -27894.149,E2 -27894.149} C_VEL
LIN {X 0,Y 92.912,Z 362.808,A -85,B 0,C 180,E1 -27902.167,E2 -27902.167} C_VEL
LIN {X 0,Y 92.534,Z 362.909,A -85,B 0,C 180,E1 -27909.819,E2 -27909.819} C_VEL
LIN {X 0,Y 94.756,Z 365.597,A -85,B 0,C 180,E1 -27921.485,E2 -27921.485} C_VEL
LIN {X 0,Y 96.553,Z 368.881,A -85,B 0,C 180,E1 -27926.185,E2 -27926.185} C_VEL
LIN {X 0,Y 97.793,Z 370.279,A -85,B 0,C 180,E1 -27928.577,E2 -27928.577} C_VEL
LIN {X 0,Y 100.715,Z 374.977,A -85,B 0,C 180,E1 -27933.422,E2 -27933.422} C_VEL
LIN {X 0,Y 104.424,Z 381.221,A -85,B 0,C 180,E1 -27938.321,E2 -27938.321} C_VEL
LIN {X 0,Y 108.619,Z 389.353,A -85,B 0,C 180,E1 -27942.932,E2 -27942.932} C_VEL
LIN {X 0,Y 111.91,Z 397.179,A -85,B 0,C 180,E1 -27946.14,E2 -27946.14} C_VEL
LIN {X 0,Y 108.347,Z 433.712,A -85,B 0,C 180,E1 -27947.833,E2 -27947.833} C_VEL
LIN {X 0,Y 105.884,Z 447.401,A -85,B 0,C 180,E1 -27949.04,E2 -27949.04} C_VEL
LIN {X 0,Y 102.876,Z 459.563,A -85,B 0,C 180,E1 -27950.801,E2 -27950.801} C_VEL
LIN {X 0,Y 99.163,Z 470.612,A -85,B 0,C 180,E1 -27952.949,E2 -27952.949} C_VEL
LIN {X 0,Y 95.038,Z 480.848,A -85,B 0,C 180,E1 -27955.669,E2 -27955.669} C_VEL
LIN {X 0,Y 91.482,Z 488.764,A -85,B 0,C 180,E1 -27958.444,E2 -27958.444} C_VEL
LIN {X 0,Y 86.251,Z 498.865,A -85,B 0,C 180,E1 -27963.105,E2 -27963.105} C_VEL
LIN {X 0,Y 81.442,Z 507.372,A -85,B 0,C 180,E1 -27968.477,E2 -27968.477} C_VEL
LIN {X 0,Y 76.754,Z 515.37,A -85,B 0,C 180,E1 -27975.408,E2 -27975.408} C_VEL
LIN {X 0,Y 73.76,Z 520.775,A -85,B 0,C 180,E1 -27981.775,E2 -27981.775} C_VEL
LIN {X 0,Y 71.22,Z 526.071,A -85,B 0,C 180,E1 -27989.992,E2 -27989.992} C_VEL
LIN {X 0,Y 69.683,Z 530.213,A -85,B 0,C 180,E1 -27998.693,E2 -27998.693} C_VEL
LIN {X 0,Y 69.397,Z 533.292,A -85,B 0,C 180,E1 -28007.678,E2 -28007.678} C_VEL
LIN {X 0,Y 70.539,Z 535.296,A -85,B 0,C 180,E1 -28016.275,E2 -28016.275} C_VEL
LIN {X 0,Y 73.186,Z 536.466,A -85,B 0,C 180,E1 -28025.171,E2 -28025.171} C_VEL
LIN {X 0,Y 77.395,Z 536.603,A -85,B 0,C 180,E1 -28033.412,E2 -28033.412} C_VEL
LIN {X 0,Y 82.407,Z 535.795,A -85,B 0,C 180,E1 -28040.122,E2 -28040.122} C_VEL
LIN {X 0,Y 88.788,Z 533.968,A -85,B 0,C 180,E1 -28046.353,E2 -28046.353} C_VEL
LIN {X 0,Y 95.862,Z 531.168,A -85,B 0,C 180,E1 -28051.599,E2 -28051.599} C_VEL
LIN {X 0,Y 103.167,Z 527.525,A -85,B 0,C 180,E1 -28055.875,E2 -28055.875} C_VEL
LIN {X 0,Y 112.143,Z 522.066,A -85,B 0,C 180,E1 -28060.042,E2 -28060.042} C_VEL
LIN {X 0,Y 121.343,Z 515.147,A -85,B 0,C 180,E1 -28063.544,E2 -28063.544} C_VEL
LIN {X 0,Y 130.206,Z 507.122,A -85,B 0,C 180,E1 -28066.283,E2 -28066.283} C_VEL
LIN {X 0,Y 138.422,Z 498.191,A -85,B 0,C 180,E1 -28068.449,E2 -28068.449} C_VEL
LIN {X 0,Y 146.165,Z 487.884,A -85,B 0,C 180,E1 -28070.267,E2 -28070.267} C_VEL
LIN {X 0,Y 153.151,Z 476.415,A -85,B 0,C 180,E1 -28071.733,E2 -28071.733} C_VEL
LIN {X 0,Y 158.24,Z 465.926,A -85,B 0,C 180,E1 -28072.762,E2 -28072.762} C_VEL
LIN {X 0,Y 162.661,Z 454.332,A -85,B 0,C 180,E1 -28073.549,E2 -28073.549} C_VEL
LIN {X 0,Y 165.982,Z 442.169,A -85,B 0,C 180,E1 -28074.198,E2 -28074.198} C_VEL
LIN {X 0,Y 165.057,Z 438.548,A -85,B 0,C 180,E1 -28077.255,E2 -28077.255} C_VEL
LIN {X 0,Y 164.33,Z 436.099,A -85,B 0,C 180,E1 -28080.001,E2 -28080.001} C_VEL
LIN {X 0,Y 163.714,Z 433.325,A -85,B 0,C 180,E1 -28084.309,E2 -28084.309} C_VEL
LIN {X 0,Y 163.565,Z 433.266,A -85,B 0,C 180,E1 -28088.818,E2 -28088.818} C_VEL
LIN {X 0,Y 163.691,Z 433.793,A -85,B 0,C 180,E1 -28090.4,E2 -28090.4} C_VEL
LIN {X 0,Y 164.665,Z 437.263,A -85,B 0,C 180,E1 -28095.63,E2 -28095.63} C_VEL
LIN {X 0,Y 165.508,Z 441.608,A -85,B 0,C 180,E1 -28098.892,E2 -28098.892} C_VEL
LIN {X 0,Y 165.848,Z 444.219,A -85,B 0,C 180,E1 -28100.387,E2 -28100.387} C_VEL
LIN {X 0,Y 162.428,Z 456.786,A -85,B 0,C 180,E1 -28100.952,E2 -28100.952} C_VEL
LIN {X 0,Y 157.847,Z 468.797,A -85,B 0,C 180,E1 -28101.664,E2 -28101.664} C_VEL
LIN {X 0,Y 152.223,Z 480.093,A -85,B 0,C 180,E1 -28102.586,E2 -28102.586} C_VEL
LIN {X 0,Y 145.815,Z 490.438,A -85,B 0,C 180,E1 -28103.698,E2 -28103.698} C_VEL
LIN {X 0,Y 138.005,Z 500.884,A -85,B 0,C 180,E1 -28105.332,E2 -28105.332} C_VEL
LIN {X 0,Y 130.388,Z 509.38,A -85,B 0,C 180,E1 -28107.219,E2 -28107.219} C_VEL
LIN {X 0,Y 121.416,Z 517.68,A -85,B 0,C 180,E1 -28109.755,E2 -28109.755} C_VEL
LIN {X 0,Y 112.775,Z 524.394,A -85,B 0,C 180,E1 -28112.733,E2 -28112.733} C_VEL
LIN {X 0,Y 104.474,Z 529.787,A -85,B 0,C 180,E1 -28116.183,E2 -28116.183} C_VEL
LIN {X 0,Y 96.788,Z 534.026,A -85,B 0,C 180,E1 -28120.331,E2 -28120.331} C_VEL
LIN {X 0,Y 89.82,Z 537.237,A -85,B 0,C 180,E1 -28125.245,E2 -28125.245} C_VEL
LIN {X 0,Y 81.605,Z 540.085,A -85,B 0,C 180,E1 -28132.935,E2 -28132.935} C_VEL
LIN {X 0,Y 75.203,Z 541.308,A -85,B 0,C 180,E1 -28142.152,E2 -28142.152} C_VEL
LIN {X 0,Y 71.314,Z 541.045,A -85,B 0,C 180,E1 -28152.812,E2 -28152.812} C_VEL
LIN {X 0,Y 70.273,Z 540.331,A -85,B 0,C 180,E1 -28158.471,E2 -28158.471} C_VEL
LIN {X 0,Y 69.878,Z 539.196,A -85,B 0,C 180,E1 -28164.236,E2 -28164.236} C_VEL
LIN {X 0,Y 69.89,Z 537.65,A -85,B 0,C 180,E1 -28170.009,E2 -28170.009} C_VEL
LIN {X 0,Y 69.985,Z 534.429,A -85,B 0,C 180,E1 -28178.672,E2 -28178.672} C_VEL
LIN {X 0,Y 71.179,Z 530.089,A -85,B 0,C 180,E1 -28187.239,E2 -28187.239} C_VEL
LIN {X 0,Y 73.728,Z 524.523,A -85,B 0,C 180,E1 -28195.41,E2 -28195.41} C_VEL
LIN {X 0,Y 77.635,Z 517.553,A -85,B 0,C 180,E1 -28202.908,E2 -28202.908} C_VEL
LIN {X 0,Y 81.539,Z 510.565,A -85,B 0,C 180,E1 -28208.5,E2 -28208.5} C_VEL
LIN {X 0,Y 86.641,Z 501.77,A -85,B 0,C 180,E1 -28213.599,E2 -28213.599} C_VEL
LIN {X 0,Y 91.454,Z 492.243,A -85,B 0,C 180,E1 -28217.711,E2 -28217.711} C_VEL
LIN {X 0,Y 94.911,Z 484.707,A -85,B 0,C 180,E1 -28220.206,E2 -28220.206} C_VEL
LIN {X 0,Y 99.269,Z 474.101,A -85,B 0,C 180,E1 -28222.804,E2 -28222.804} C_VEL
LIN {X 0,Y 103.126,Z 462.427,A -85,B 0,C 180,E1 -28224.874,E2 -28224.874} C_VEL
LIN {X 0,Y 106.405,Z 449.197,A -85,B 0,C 180,E1 -28226.508,E2 -28226.508} C_VEL
LIN {X 0,Y 108.494,Z 436.568,A -85,B 0,C 180,E1 -28227.495,E2 -28227.495} C_VEL
LIN {X 0,Y 111.498,Z 403.462,A -85,B 0,C 180,E1 -28229.083,E2 -28229.083} C_VEL
LIN {X 0,Y 111.334,Z 400.346,A -85,B 0,C 180,E1 -28229.519,E2 -28229.519} C_VEL
LIN {X 0,Y 110.216,Z 396.913,A -85,B 0,C 180,E1 -28230.656,E2 -28230.656} C_VEL
LIN {X 0,Y 107.872,Z 393.303,A -85,B 0,C 180,E1 -28232.803,E2 -28232.803} C_VEL
LIN {X 0,Y 101.535,Z 386.49,A -85,B 0,C 180,E1 -28239.454,E2 -28239.454} C_VEL
LIN {X 0,Y 100.199,Z 383.923,A -85,B 0,C 180,E1 -28241.338,E2 -28241.338} C_VEL
LIN {X 0,Y 97.6,Z 379.32,A -85,B 0,C 180,E1 -28245.505,E2 -28245.505} C_VEL
LIN {X 0,Y 95.749,Z 376.115,A -85,B 0,C 180,E1 -28249.158,E2 -28249.158} C_VEL
LIN {X 0,Y 93.766,Z 372.646,A -85,B 0,C 180,E1 -28254.337,E2 -28254.337} C_VEL
LIN {X 0,Y 93.379,Z 371.837,A -85,B 0,C 180,E1 -28255.683,E2 -28255.683} C_VEL
LIN {X 0,Y 92.022,Z 369.866,A -85,B 0,C 180,E1 -28262.188,E2 -28262.188} C_VEL
LIN {X 0,Y 91.635,Z 369.809,A -85,B 0,C 180,E1 -28268.823,E2 -28268.823} C_VEL
LIN {X 0,Y 93.461,Z 372.427,A -85,B 0,C 180,E1 -28280.372,E2 -28280.372} C_VEL
LIN {X 0,Y 95.208,Z 375.73,A -85,B 0,C 180,E1 -28285.354,E2 -28285.354} C_VEL
LIN {X 0,Y 96.137,Z 376.989,A -85,B 0,C 180,E1 -28287.334,E2 -28287.334} C_VEL
LIN {X 0,Y 98.698,Z 381.379,A -85,B 0,C 180,E1 -28292.003,E2 -28292.003} C_VEL
LIN {X 0,Y 101.833,Z 387,A -85,B 0,C 180,E1 -28296.553,E2 -28296.553} C_VEL
LIN {X 0,Y 105.434,Z 394.546,A -85,B 0,C 180,E1 -28300.988,E2 -28300.988} C_VEL
LIN {X 0,Y 107.38,Z 399.424,A -85,B 0,C 180,E1 -28303.156,E2 -28303.156} C_VEL
LIN {X 0,Y 104.029,Z 433.553,A -85,B 0,C 180,E1 -28304.795,E2 -28304.795} C_VEL
LIN {X 0,Y 101.473,Z 447.25,A -85,B 0,C 180,E1 -28305.961,E2 -28305.961} C_VEL
LIN {X 0,Y 98.119,Z 460.118,A -85,B 0,C 180,E1 -28307.809,E2 -28307.809} C_VEL
LIN {X 0,Y 94.205,Z 471.109,A -85,B 0,C 180,E1 -28309.942,E2 -28309.942} C_VEL
LIN {X 0,Y 89.849,Z 481.301,A -85,B 0,C 180,E1 -28312.677,E2 -28312.677} C_VEL
LIN {X 0,Y 85.597,Z 489.985,A -85,B 0,C 180,E1 -28315.802,E2 -28315.802} C_VEL
LIN {X 0,Y 80.803,Z 498.718,A -85,B 0,C 180,E1 -28319.984,E2 -28319.984} C_VEL
LIN {X 0,Y 75.783,Z 506.991,A -85,B 0,C 180,E1 -28325.326,E2 -28325.326} C_VEL
LIN {X 0,Y 70.614,Z 515.109,A -85,B 0,C 180,E1 -28332.619,E2 -28332.619} C_VEL
LIN {X 0,Y 66.684,Z 521.605,A -85,B 0,C 180,E1 -28340.895,E2 -28340.895} C_VEL
LIN {X 0,Y 63.985,Z 526.769,A -85,B 0,C 180,E1 -28349.991,E2 -28349.991} C_VEL
LIN {X 0,Y 62.457,Z 530.807,A -85,B 0,C 180,E1 -28359.707,E2 -28359.707} C_VEL
LIN {X 0,Y 62.424,Z 533.791,A -85,B 0,C 180,E1 -28369.73,E2 -28369.73} C_VEL
LIN {X 0,Y 63.718,Z 535.526,A -85,B 0,C 180,E1 -28378.07,E2 -28378.07} C_VEL
LIN {X 0,Y 67.226,Z 536.799,A -85,B 0,C 180,E1 -28388.836,E2 -28388.836} C_VEL
LIN {X 0,Y 71.483,Z 536.879,A -85,B 0,C 180,E1 -28396.512,E2 -28396.512} C_VEL
LIN {X 0,Y 77.82,Z 535.951,A -85,B 0,C 180,E1 -28404.356,E2 -28404.356} C_VEL
LIN {X 0,Y 83.934,Z 534.306,A -85,B 0,C 180,E1 -28409.843,E2 -28409.843} C_VEL
LIN {X 0,Y 92.539,Z 531.125,A -85,B 0,C 180,E1 -28415.676,E2 -28415.676} C_VEL
LIN {X 0,Y 101.237,Z 526.918,A -85,B 0,C 180,E1 -28420.152,E2 -28420.152} C_VEL
LIN {X 0,Y 111.347,Z 520.735,A -85,B 0,C 180,E1 -28424.248,E2 -28424.248} C_VEL
LIN {X 0,Y 120.487,Z 513.869,A -85,B 0,C 180,E1 -28427.284,E2 -28427.284} C_VEL
LIN {X 0,Y 128.652,Z 506.549,A -85,B 0,C 180,E1 -28429.487,E2 -28429.487} C_VEL
LIN {X 0,Y 136.809,Z 497.777,A -85,B 0,C 180,E1 -28431.416,E2 -28431.416} C_VEL
LIN {X 0,Y 144.263,Z 488.04,A -85,B 0,C 180,E1 -28432.986,E2 -28432.986} C_VEL
LIN {X 0,Y 151.016,Z 477.261,A -85,B 0,C 180,E1 -28434.262,E2 -28434.262} C_VEL
LIN {X 0,Y 156.895,Z 465.436,A -85,B 0,C 180,E1 -28435.328,E2 -28435.328} C_VEL
LIN {X 0,Y 161.548,Z 453.083,A -85,B 0,C 180,E1 -28436.075,E2 -28436.075} C_VEL
LIN {X 0,Y 163.395,Z 446.718,A -85,B 0,C 180,E1 -28436.425,E2 -28436.425} C_VEL
LIN {X 0,Y 162.827,Z 443.601,A -85,B 0,C 180,E1 -28439.537,E2 -28439.537} C_VEL
LIN {X 0,Y 162.309,Z 440.193,A -85,B 0,C 180,E1 -28444.969,E2 -28444.969} C_VEL
LIN {X 0,Y 162.312,Z 440.348,A -85,B 0,C 180,E1 -28449.43,E2 -28449.43} C_VEL
LIN {X 0,Y 162.943,Z 443.938,A -85,B 0,C 180,E1 -28454.999,E2 -28454.999} C_VEL
LIN {X 0,Y 163.361,Z 447.937,A -85,B 0,C 180,E1 -28457.991,E2 -28457.991} C_VEL
LIN {X 0,Y 163.212,Z 448.774,A -85,B 0,C 180,E1 -28458.163,E2 -28458.163} C_VEL
LIN {X 0,Y 159.041,Z 461.696,A -85,B 0,C 180,E1 -28458.732,E2 -28458.732} C_VEL
LIN {X 0,Y 153.752,Z 473.771,A -85,B 0,C 180,E1 -28459.492,E2 -28459.492} C_VEL
LIN {X 0,Y 147.193,Z 485.314,A -85,B 0,C 180,E1 -28460.455,E2 -28460.455} C_VEL
LIN {X 0,Y 140.749,Z 494.639,A -85,B 0,C 180,E1 -28461.578,E2 -28461.578} C_VEL
LIN {X 0,Y 133.542,Z 503.341,A -85,B 0,C 180,E1 -28462.943,E2 -28462.943} C_VEL
LIN {X 0,Y 124.161,Z 512.82,A -85,B 0,C 180,E1 -28465.1,E2 -28465.1} C_VEL
LIN {X 0,Y 115.049,Z 520.389,A -85,B 0,C 180,E1 -28467.667,E2 -28467.667} C_VEL
LIN {X 0,Y 106.182,Z 526.514,A -85,B 0,C 180,E1 -28470.645,E2 -28470.645} C_VEL
LIN {X 0,Y 97.673,Z 531.407,A -85,B 0,C 180,E1 -28474.172,E2 -28474.172} C_VEL
LIN {X 0,Y 89.789,Z 535.208,A -85,B 0,C 180,E1 -28478.501,E2 -28478.501} C_VEL
LIN {X 0,Y 80.306,Z 538.769,A -85,B 0,C 180,E1 -28485.575,E2 -28485.575} C_VEL
LIN {X 0,Y 76.038,Z 539.926,A -85,B 0,C 180,E1 -28489.695,E2 -28489.695} C_VEL
LIN {X 0,Y 68.98,Z 541.062,A -85,B 0,C 180,E1 -28499.385,E2 -28499.385} C_VEL
LIN {X 0,Y 64.536,Z 540.713,A -85,B 0,C 180,E1 -28510.941,E2 -28510.941} C_VEL
LIN {X 0,Y 62.831,Z 538.755,A -85,B 0,C 180,E1 -28523.587,E2 -28523.587} C_VEL
LIN {X 0,Y 62.817,Z 537.17,A -85,B 0,C 180,E1 -28530.01,E2 -28530.01} C_VEL
LIN {X 0,Y 62.964,Z 533.861,A -85,B 0,C 180,E1 -28539.648,E2 -28539.648} C_VEL
LIN {X 0,Y 64.399,Z 529.429,A -85,B 0,C 180,E1 -28549.12,E2 -28549.12} C_VEL
LIN {X 0,Y 67.365,Z 523.766,A -85,B 0,C 180,E1 -28558.01,E2 -28558.01} C_VEL
LIN {X 0,Y 71.711,Z 516.648,A -85,B 0,C 180,E1 -28566.027,E2 -28566.027} C_VEL
LIN {X 0,Y 75.226,Z 510.905,A -85,B 0,C 180,E1 -28570.852,E2 -28570.852} C_VEL
LIN {X 0,Y 78.318,Z 506.018,A -85,B 0,C 180,E1 -28574.117,E2 -28574.117} C_VEL
LIN {X 0,Y 83.793,Z 496.455,A -85,B 0,C 180,E1 -28579.023,E2 -28579.023} C_VEL
LIN {X 0,Y 88.548,Z 487.073,A -85,B 0,C 180,E1 -28582.542,E2 -28582.542} C_VEL
LIN {X 0,Y 93.818,Z 475.539,A -85,B 0,C 180,E1 -28585.5,E2 -28585.5} C_VEL
LIN {X 0,Y 97.113,Z 466.436,A -85,B 0,C 180,E1 -28587.287,E2 -28587.287} C_VEL
LIN {X 0,Y 100.939,Z 453.41,A -85,B 0,C 180,E1 -28589.079,E2 -28589.079} C_VEL
LIN {X 0,Y 103.541,Z 440.348,A -85,B 0,C 180,E1 -28590.245,E2 -28590.245} C_VEL
LIN {X 0,Y 105.626,Z 421.664,A -85,B 0,C 180,E1 -28591.193,E2 -28591.193} C_VEL
LIN {X 0,Y 107.289,Z 402.34,A -85,B 0,C 180,E1 -28592.178,E2 -28592.178} C_VEL
LIN {X 0,Y 105.063,Z 393.968,A -85,B 0,C 180,E1 -28595.007,E2 -28595.007} C_VEL
LIN {X 0,Y 101.692,Z 386.719,A -85,B 0,C 180,E1 -28599.238,E2 -28599.238} C_VEL
LIN {X 0,Y 100.199,Z 383.923,A -85,B 0,C 180,E1 -28601.338,E2 -28601.338} C_VEL
LIN {X 0,Y 99.057,Z 381.773,A -85,B 0,C 180,E1 -28603.082,E2 -28603.082} C_VEL
LIN {X 0,Y 97.115,Z 379.829,A -85,B 0,C 180,E1 -28606.117,E2 -28606.117} C_VEL
LIN {X 0,Y 95.216,Z 378.989,A -85,B 0,C 180,E1 -28609.439,E2 -28609.439} C_VEL
LIN {X 0,Y 92.167,Z 378.463,A -85,B 0,C 180,E1 -28616.807,E2 -28616.807} C_VEL
LIN {X 0,Y 91.544,Z 378,A -85,B 0,C 180,E1 -28619.341,E2 -28619.341} C_VEL
LIN {X 0,Y 90.994,Z 376.826,A -85,B 0,C 180,E1 -28623.328,E2 -28623.328} C_VEL
LIN {X 0,Y 90.776,Z 377.092,A -85,B 0,C 180,E1 -28630.122,E2 -28630.122} C_VEL
LIN {X 0,Y 92.195,Z 379.267,A -85,B 0,C 180,E1 -28639.209,E2 -28639.209} C_VEL
LIN {X 0,Y 93.999,Z 382.682,A -85,B 0,C 180,E1 -28644.762,E2 -28644.762} C_VEL
LIN {X 0,Y 96.514,Z 387.296,A -85,B 0,C 180,E1 -28650.097,E2 -28650.097} C_VEL
LIN {X 0,Y 99.366,Z 392.932,A -85,B 0,C 180,E1 -28654.77,E2 -28654.77} C_VEL
LIN {X 0,Y 102.369,Z 399.829,A -85,B 0,C 180,E1 -28658.928,E2 -28658.928} C_VEL
LIN {X 0,Y 103.241,Z 402.239,A -85,B 0,C 180,E1 -28660.061,E2 -28660.061} C_VEL
LIN {X 0,Y 100.08,Z 433.098,A -85,B 0,C 180,E1 -28661.489,E2 -28661.489} C_VEL
LIN {X 0,Y 97.472,Z 446.712,A -85,B 0,C 180,E1 -28662.574,E2 -28662.574} C_VEL
LIN {X 0,Y 93.984,Z 459.668,A -85,B 0,C 180,E1 -28664.342,E2 -28664.342} C_VEL
LIN {X 0,Y 89.534,Z 471.606,A -85,B 0,C 180,E1 -28666.612,E2 -28666.612} C_VEL
LIN {X 0,Y 84.318,Z 483.045,A -85,B 0,C 180,E1 -28669.753,E2 -28669.753} C_VEL
LIN {X 0,Y 79.669,Z 491.679,A -85,B 0,C 180,E1 -28672.991,E2 -28672.991} C_VEL
LIN {X 0,Y 74.711,Z 500.011,A -85,B 0,C 180,E1 -28677.246,E2 -28677.246} C_VEL
LIN {X 0,Y 69.345,Z 508.117,A -85,B 0,C 180,E1 -28682.857,E2 -28682.857} C_VEL
LIN {X 0,Y 63.801,Z 516.066,A -85,B 0,C 180,E1 -28690.693,E2 -28690.693} C_VEL
LIN {X 0,Y 59.592,Z 522.399,A -85,B 0,C 180,E1 -28699.8,E2 -28699.8} C_VEL
LIN {X 0,Y 56.736,Z 527.456,A -85,B 0,C 180,E1 -28709.989,E2 -28709.989} C_VEL
LIN {X 0,Y 55.25,Z 531.395,A -85,B 0,C 180,E1 -28720.989,E2 -28720.989} C_VEL
LIN {X 0,Y 55.557,Z 534.28,A -85,B 0,C 180,E1 -28732.291,E2 -28732.291} C_VEL
LIN {X 0,Y 56.97,Z 535.755,A -85,B 0,C 180,E1 -28740.287,E2 -28740.287} C_VEL
LIN {X 0,Y 58.824,Z 536.607,A -85,B 0,C 180,E1 -28746.669,E2 -28746.669} C_VEL
LIN {X 0,Y 61.603,Z 537.101,A -85,B 0,C 180,E1 -28753.183,E2 -28753.183} C_VEL
LIN {X 0,Y 65.848,Z 537.154,A -85,B 0,C 180,E1 -28760.181,E2 -28760.181} C_VEL
LIN {X 0,Y 73.712,Z 536.079,A -85,B 0,C 180,E1 -28769.086,E2 -28769.086} C_VEL
LIN {X 0,Y 79.447,Z 534.644,A -85,B 0,C 180,E1 -28773.75,E2 -28773.75} C_VEL
LIN {X 0,Y 89.727,Z 531.069,A -85,B 0,C 180,E1 -28780.016,E2 -28780.016} C_VEL
LIN {X 0,Y 98.344,Z 527.07,A -85,B 0,C 180,E1 -28783.96,E2 -28783.96} C_VEL
LIN {X 0,Y 107.971,Z 521.472,A -85,B 0,C 180,E1 -28787.493,E2 -28787.493} C_VEL
LIN {X 0,Y 117.602,Z 514.586,A -85,B 0,C 180,E1 -28790.385,E2 -28790.385} C_VEL
LIN {X 0,Y 125.843,Z 507.512,A -85,B 0,C 180,E1 -28792.392,E2 -28792.392} C_VEL
LIN {X 0,Y 134.216,Z 498.919,A -85,B 0,C 180,E1 -28794.163,E2 -28794.163} C_VEL
LIN {X 0,Y 141.842,Z 489.414,A -85,B 0,C 180,E1 -28795.613,E2 -28795.613} C_VEL
LIN {X 0,Y 148.9,Z 478.594,A -85,B 0,C 180,E1 -28796.808,E2 -28796.808} C_VEL
LIN {X 0,Y 154.722,Z 467.427,A -85,B 0,C 180,E1 -28797.76,E2 -28797.76} C_VEL
LIN {X 0,Y 159.385,Z 456.004,A -85,B 0,C 180,E1 -28798.421,E2 -28798.421} C_VEL
LIN {X 0,Y 160.845,Z 451.423,A -85,B 0,C 180,E1 -28798.747,E2 -28798.747} C_VEL
LIN {X 0,Y 160.5,Z 448.701,A -85,B 0,C 180,E1 -28802.51,E2 -28802.51} C_VEL
LIN {X 0,Y 160.551,Z 447.102,A -85,B 0,C 180,E1 -28805.023,E2 -28805.023} C_VEL
LIN {X 0,Y 160.564,Z 447.179,A -85,B 0,C 180,E1 -28809.13,E2 -28809.13} C_VEL
LIN {X 0,Y 160.886,Z 450.561,A -85,B 0,C 180,E1 -28814.386,E2 -28814.386} C_VEL
LIN {X 0,Y 160.937,Z 451.481,A -85,B 0,C 180,E1 -28815.19,E2 -28815.19} C_VEL
LIN {X 0,Y 160.722,Z 453.033,A -85,B 0,C 180,E1 -28815.86,E2 -28815.86} C_VEL
LIN {X 0,Y 156.248,Z 465.222,A -85,B 0,C 180,E1 -28816.403,E2 -28816.403} C_VEL
LIN {X 0,Y 150.713,Z 476.696,A -85,B 0,C 180,E1 -28817.085,E2 -28817.085} C_VEL
LIN {X 0,Y 144.046,Z 487.64,A -85,B 0,C 180,E1 -28817.951,E2 -28817.951} C_VEL
LIN {X 0,Y 137.486,Z 496.524,A -85,B 0,C 180,E1 -28818.987,E2 -28818.987} C_VEL
LIN {X 0,Y 130.954,Z 503.99,A -85,B 0,C 180,E1 -28820.1,E2 -28820.1} C_VEL
LIN {X 0,Y 122.954,Z 511.852,A -85,B 0,C 180,E1 -28821.76,E2 -28821.76} C_VEL
LIN {X 0,Y 113.504,Z 519.583,A -85,B 0,C 180,E1 -28824.05,E2 -28824.05} C_VEL
LIN {X 0,Y 102.754,Z 526.715,A -85,B 0,C 180,E1 -28827.247,E2 -28827.247} C_VEL
LIN {X 0,Y 93.873,Z 531.505,A -85,B 0,C 180,E1 -28830.588,E2 -28830.588} C_VEL
LIN {X 0,Y 85.54,Z 535.209,A -85,B 0,C 180,E1 -28834.768,E2 -28834.768} C_VEL
LIN {X 0,Y 80.315,Z 537.144,A -85,B 0,C 180,E1 -28838.056,E2 -28838.056} C_VEL
LIN {X 0,Y 75.394,Z 538.666,A -85,B 0,C 180,E1 -28841.79,E2 -28841.79} C_VEL
LIN {X 0,Y 66.607,Z 540.474,A -85,B 0,C 180,E1 -28850.734,E2 -28850.734} C_VEL
LIN {X 0,Y 60.041,Z 540.79,A -85,B 0,C 180,E1 -28862.093,E2 -28862.093} C_VEL
LIN {X 0,Y 56.421,Z 539.527,A -85,B 0,C 180,E1 -28875.585,E2 -28875.585} C_VEL
LIN {X 0,Y 55.776,Z 538.314,A -85,B 0,C 180,E1 -28882.772,E2 -28882.772} C_VEL
LIN {X 0,Y 55.715,Z 536.688,A -85,B 0,C 180,E1 -28890.011,E2 -28890.011} C_VEL
LIN {X 0,Y 55.946,Z 533.292,A -85,B 0,C 180,E1 -28900.872,E2 -28900.872} C_VEL
LIN {X 0,Y 57.675,Z 528.766,A -85,B 0,C 180,E1 -28911.453,E2 -28911.453} C_VEL
LIN {X 0,Y 61.162,Z 522.997,A -85,B 0,C 180,E1 -28921.148,E2 -28921.148} C_VEL
LIN {X 0,Y 66.054,Z 515.716,A -85,B 0,C 180,E1 -28929.683,E2 -28929.683} C_VEL
LIN {X 0,Y 69.901,Z 509.897,A -85,B 0,C 180,E1 -28934.743,E2 -28934.743} C_VEL
LIN {X 0,Y 75.711,Z 501.3,A -85,B 0,C 180,E1 -28939.991,E2 -28939.991} C_VEL
LIN {X 0,Y 81.218,Z 491.785,A -85,B 0,C 180,E1 -28944.229,E2 -28944.229} C_VEL
LIN {X 0,Y 85.11,Z 484.255,A -85,B 0,C 180,E1 -28946.74,E2 -28946.74} C_VEL
LIN {X 0,Y 89.936,Z 473.673,A -85,B 0,C 180,E1 -28949.282,E2 -28949.282} C_VEL
LIN {X 0,Y 94.188,Z 462.033,A -85,B 0,C 180,E1 -28951.265,E2 -28951.265} C_VEL
LIN {X 0,Y 97.806,Z 448.661,A -85,B 0,C 180,E1 -28952.852,E2 -28952.852} C_VEL
LIN {X 0,Y 100.14,Z 435.495,A -85,B 0,C 180,E1 -28953.818,E2 -28953.818} C_VEL
LIN {X 0,Y 103.237,Z 404.549,A -85,B 0,C 180,E1 -28955.239,E2 -28955.239} C_VEL
LIN {X 0,Y 101.612,Z 398.107,A -85,B 0,C 180,E1 -28957.65,E2 -28957.65} C_VEL
LIN {X 0,Y 98.663,Z 391.429,A -85,B 0,C 180,E1 -28961.921,E2 -28961.921} C_VEL
LIN {X 0,Y 95.91,Z 385.907,A -85,B 0,C 180,E1 -28966.714,E2 -28966.714} C_VEL
LIN {X 0,Y 94.044,Z 382.549,A -85,B 0,C 180,E1 -28970.794,E2 -28970.794} C_VEL
LIN {X 0,Y 92.166,Z 378.681,A -85,B 0,C 180,E1 -28976.721,E2 -28976.721} C_VEL
LIN {X 0,Y 91.544,Z 378,A -85,B 0,C 180,E1 -28979.341,E2 -28979.341} C_VEL
LIN {X 0,Y 90.902,Z 377.87,A -85,B 0,C 180,E1 -28983.028,E2 -28983.028} C_VEL
LIN {X 0,Y 90.482,Z 378.995,A -85,B 0,C 180,E1 -28986.712,E2 -28986.712} C_VEL
LIN {X 0,Y 90.313,Z 381.718,A -85,B 0,C 180,E1 -28991.532,E2 -28991.532} C_VEL
LIN {X 0,Y 91.107,Z 386.504,A -85,B 0,C 180,E1 -28998.671,E2 -28998.671} C_VEL
LIN {X 0,Y 92.943,Z 390.176,A -85,B 0,C 180,E1 -29004.604,E2 -29004.604} C_VEL
LIN {X 0,Y 94.736,Z 393.887,A -85,B 0,C 180,E1 -29008.732,E2 -29008.732} C_VEL
LIN {X 0,Y 97.446,Z 399.925,A -85,B 0,C 180,E1 -29013.65,E2 -29013.65} C_VEL
LIN {X 0,Y 99.415,Z 404.985,A -85,B 0,C 180,E1 -29016.695,E2 -29016.695} C_VEL
LIN {X 0,Y 96.262,Z 434.008,A -85,B 0,C 180,E1 -29018.006,E2 -29018.006} C_VEL
LIN {X 0,Y 93.451,Z 447.796,A -85,B 0,C 180,E1 -29019.074,E2 -29019.074} C_VEL
LIN {X 0,Y 89.877,Z 460.234,A -85,B 0,C 180,E1 -29020.744,E2 -29020.744} C_VEL
LIN {X 0,Y 85.188,Z 472.109,A -85,B 0,C 180,E1 -29022.92,E2 -29022.92} C_VEL
LIN {X 0,Y 79.69,Z 483.498,A -85,B 0,C 180,E1 -29026.002,E2 -29026.002} C_VEL
LIN {X 0,Y 73.881,Z 493.543,A -85,B 0,C 180,E1 -29029.838,E2 -29029.838} C_VEL
LIN {X 0,Y 67.622,Z 502.995,A -85,B 0,C 180,E1 -29035.127,E2 -29035.127} C_VEL
LIN {X 0,Y 60.909,Z 512.003,A -85,B 0,C 180,E1 -29042.502,E2 -29042.502} C_VEL
LIN {X 0,Y 55.406,Z 519.231,A -85,B 0,C 180,E1 -29051.5,E2 -29051.5} C_VEL
LIN {X 0,Y 51.326,Z 524.991,A -85,B 0,C 180,E1 -29062.118,E2 -29062.118} C_VEL
LIN {X 0,Y 48.838,Z 529.483,A -85,B 0,C 180,E1 -29073.889,E2 -29073.889} C_VEL
LIN {X 0,Y 48.057,Z 533.035,A -85,B 0,C 180,E1 -29086.994,E2 -29086.994} C_VEL
LIN {X 0,Y 50.297,Z 535.971,A -85,B 0,C 180,E1 -29103.034,E2 -29103.034} C_VEL
LIN {X 0,Y 53.045,Z 536.966,A -85,B 0,C 180,E1 -29111.472,E2 -29111.472} C_VEL
LIN {X 0,Y 56.395,Z 537.402,A -85,B 0,C 180,E1 -29118.377,E2 -29118.377} C_VEL
LIN {X 0,Y 60.512,Z 537.43,A -85,B 0,C 180,E1 -29124.501,E2 -29124.501} C_VEL
LIN {X 0,Y 65.08,Z 537.05,A -85,B 0,C 180,E1 -29129.741,E2 -29129.741} C_VEL
LIN {X 0,Y 70.176,Z 536.196,A -85,B 0,C 180,E1 -29134.313,E2 -29134.313} C_VEL
LIN {X 0,Y 75.648,Z 534.918,A -85,B 0,C 180,E1 -29138.262,E2 -29138.262} C_VEL
LIN {X 0,Y 84.412,Z 532.149,A -85,B 0,C 180,E1 -29143.202,E2 -29143.202} C_VEL
LIN {X 0,Y 93.689,Z 528.277,A -85,B 0,C 180,E1 -29147.176,E2 -29147.176} C_VEL
LIN {X 0,Y 103.331,Z 523.187,A -85,B 0,C 180,E1 -29150.434,E2 -29150.434} C_VEL
LIN {X 0,Y 113.236,Z 516.697,A -85,B 0,C 180,E1 -29153.184,E2 -29153.184} C_VEL
LIN {X 0,Y 123.373,Z 508.477,A -85,B 0,C 180,E1 -29155.411,E2 -29155.411} C_VEL
LIN {X 0,Y 132.595,Z 499.326,A -85,B 0,C 180,E1 -29157.131,E2 -29157.131} C_VEL
LIN {X 0,Y 140.599,Z 489.574,A -85,B 0,C 180,E1 -29158.459,E2 -29158.459} C_VEL
LIN {X 0,Y 147.581,Z 479.09,A -85,B 0,C 180,E1 -29159.499,E2 -29159.499} C_VEL
LIN {X 0,Y 154.028,Z 466.91,A -85,B 0,C 180,E1 -29160.417,E2 -29160.417} C_VEL
LIN {X 0,Y 158.272,Z 456.574,A -85,B 0,C 180,E1 -29160.954,E2 -29160.954} C_VEL
LIN {X 0,Y 158.376,Z 454.041,A -85,B 0,C 180,E1 -29165.092,E2 -29165.092} C_VEL
LIN {X 0,Y 158.405,Z 453.764,A -85,B 0,C 180,E1 -29167.649,E2 -29167.649} C_VEL
LIN {X 0,Y 158.335,Z 454.831,A -85,B 0,C 180,E1 -29170.228,E2 -29170.228} C_VEL
LIN {X 0,Y 158.492,Z 456.488,A -85,B 0,C 180,E1 -29173.15,E2 -29173.15} C_VEL
LIN {X 0,Y 158.021,Z 458.075,A -85,B 0,C 180,E1 -29173.521,E2 -29173.521} C_VEL
LIN {X 0,Y 152.732,Z 470.514,A -85,B 0,C 180,E1 -29174.064,E2 -29174.064} C_VEL
LIN {X 0,Y 146.26,Z 482.262,A -85,B 0,C 180,E1 -29174.771,E2 -29174.771} C_VEL
LIN {X 0,Y 138.674,Z 493.124,A -85,B 0,C 180,E1 -29175.67,E2 -29175.67} C_VEL
LIN {X 0,Y 130.355,Z 502.866,A -85,B 0,C 180,E1 -29176.885,E2 -29176.885} C_VEL
LIN {X 0,Y 122.164,Z 510.867,A -85,B 0,C 180,E1 -29178.353,E2 -29178.353} C_VEL
LIN {X 0,Y 114.008,Z 517.539,A -85,B 0,C 180,E1 -29179.952,E2 -29179.952} C_VEL
LIN {X 0,Y 106.01,Z 523.117,A -85,B 0,C 180,E1 -29181.87,E2 -29181.87} C_VEL
LIN {X 0,Y 96.581,Z 528.595,A -85,B 0,C 180,E1 -29184.567,E2 -29184.567} C_VEL
LIN {X 0,Y 87.493,Z 532.915,A -85,B 0,C 180,E1 -29187.938,E2 -29187.938} C_VEL
LIN {X 0,Y 77.441,Z 536.667,A -85,B 0,C 180,E1 -29192.993,E2 -29192.993} C_VEL
LIN {X 0,Y 70.842,Z 538.547,A -85,B 0,C 180,E1 -29197.487,E2 -29197.487} C_VEL
LIN {X 0,Y 61.265,Z 540.269,A -85,B 0,C 180,E1 -29206.52,E2 -29206.52} C_VEL
LIN {X 0,Y 57.187,Z 540.571,A -85,B 0,C 180,E1 -29212.1,E2 -29212.1} C_VEL
LIN {X 0,Y 53.835,Z 540.481,A -85,B 0,C 180,E1 -29218.534,E2 -29218.534} C_VEL
LIN {X 0,Y 49.572,Z 539.126,A -85,B 0,C 180,E1 -29233.541,E2 -29233.541} C_VEL
LIN {X 0,Y 48.751,Z 537.874,A -85,B 0,C 180,E1 -29241.724,E2 -29241.724} C_VEL
LIN {X 0,Y 48.629,Z 536.194,A -85,B 0,C 180,E1 -29250.012,E2 -29250.012} C_VEL
LIN {X 0,Y 48.974,Z 532.716,A -85,B 0,C 180,E1 -29262.443,E2 -29262.443} C_VEL
LIN {X 0,Y 51.083,Z 528.088,A -85,B 0,C 180,E1 -29274.389,E2 -29274.389} C_VEL
LIN {X 0,Y 56.027,Z 521.061,A -85,B 0,C 180,E1 -29286.585,E2 -29286.585} C_VEL
LIN {X 0,Y 61.808,Z 513.416,A -85,B 0,C 180,E1 -29295.302,E2 -29295.302} C_VEL
LIN {X 0,Y 66.189,Z 507.281,A -85,B 0,C 180,E1 -29300.263,E2 -29300.263} C_VEL
LIN {X 0,Y 71.3,Z 500.069,A -85,B 0,C 180,E1 -29304.423,E2 -29304.423} C_VEL
LIN {X 0,Y 77.244,Z 490.364,A -85,B 0,C 180,E1 -29308.551,E2 -29308.551} C_VEL
LIN {X 0,Y 81.443,Z 482.653,A -85,B 0,C 180,E1 -29310.908,E2 -29310.908} C_VEL
LIN {X 0,Y 86.466,Z 471.654,A -85,B 0,C 180,E1 -29313.406,E2 -29313.406} C_VEL
LIN {X 0,Y 90.94,Z 459.535,A -85,B 0,C 180,E1 -29315.253,E2 -29315.253} C_VEL
LIN {X 0,Y 94.385,Z 446.821,A -85,B 0,C 180,E1 -29316.569,E2 -29316.569} C_VEL
LIN {X 0,Y 96.711,Z 433.102,A -85,B 0,C 180,E1 -29317.455,E2 -29317.455} C_VEL
LIN {X 0,Y 99.46,Z 406.645,A -85,B 0,C 180,E1 -29318.604,E2 -29318.604} C_VEL
LIN {X 0,Y 98.502,Z 402.648,A -85,B 0,C 180,E1 -29320.28,E2 -29320.28} C_VEL
LIN {X 0,Y 96.223,Z 397.03,A -85,B 0,C 180,E1 -29324.062,E2 -29324.062} C_VEL
LIN {X 0,Y 93.913,Z 391.944,A -85,B 0,C 180,E1 -29328.704,E2 -29328.704} C_VEL
LIN {X 0,Y 92.435,Z 388.958,A -85,B 0,C 180,E1 -29332.456,E2 -29332.456} C_VEL
LIN {X 0,Y 90.987,Z 385.508,A -85,B 0,C 180,E1 -29337.786,E2 -29337.786} C_VEL
LIN {X 0,Y 90.108,Z 383.854,A -85,B 0,C 180,E1 -29343.36,E2 -29343.36} C_VEL
LIN {X 0,Y 89.886,Z 384.247,A -85,B 0,C 180,E1 -29350.223,E2 -29350.223} C_VEL
LIN {X 0,Y 90.997,Z 386.132,A -85,B 0,C 180,E1 -29358.132,E2 -29358.132} C_VEL
LIN {X 0,Y 91.107,Z 386.504,A -85,B 0,C 180,E1 -29358.671,E2 -29358.671} C_VEL
LIN {X 0,Y 91.883,Z 389.254,A -85,B 0,C 180,E1 -29361.92,E2 -29361.92} C_VEL
LIN {X 0,Y 92.664,Z 392.96,A -85,B 0,C 180,E1 -29364.777,E2 -29364.777} C_VEL
LIN {X 0,Y 95.822,Z 407.774,A -85,B 0,C 180,E1 -29372.976,E2 -29372.976} C_VEL
LIN {X 0,Y 95.918,Z 408.268,A -85,B 0,C 180,E1 -29373.185,E2 -29373.185} C_VEL
LIN {X 0,Y 92.859,Z 434.534,A -85,B 0,C 180,E1 -29374.248,E2 -29374.248} C_VEL
LIN {X 0,Y 89.933,Z 448.225,A -85,B 0,C 180,E1 -29375.229,E2 -29375.229} C_VEL
LIN {X 0,Y 86.157,Z 460.69,A -85,B 0,C 180,E1 -29376.819,E2 -29376.819} C_VEL
LIN {X 0,Y 81.235,Z 472.53,A -85,B 0,C 180,E1 -29378.854,E2 -29378.854} C_VEL
LIN {X 0,Y 75.445,Z 483.888,A -85,B 0,C 180,E1 -29381.81,E2 -29381.81} C_VEL
LIN {X 0,Y 69.797,Z 493.092,A -85,B 0,C 180,E1 -29385.172,E2 -29385.172} C_VEL
LIN {X 0,Y 63.18,Z 502.519,A -85,B 0,C 180,E1 -29390.225,E2 -29390.225} C_VEL
LIN {X 0,Y 55.812,Z 511.646,A -85,B 0,C 180,E1 -29397.632,E2 -29397.632} C_VEL
LIN {X 0,Y 49.561,Z 518.999,A -85,B 0,C 180,E1 -29407.035,E2 -29407.035} C_VEL
LIN {X 0,Y 45.512,Z 523.965,A -85,B 0,C 180,E1 -29416.593,E2 -29416.593} C_VEL
LIN {X 0,Y 42.168,Z 528.96,A -85,B 0,C 180,E1 -29430.468,E2 -29430.468} C_VEL
LIN {X 0,Y 40.951,Z 532.556,A -85,B 0,C 180,E1 -29444.902,E2 -29444.902} C_VEL
LIN {X 0,Y 42.252,Z 535.25,A -85,B 0,C 180,E1 -29459.917,E2 -29459.917} C_VEL
LIN {X 0,Y 44.532,Z 536.513,A -85,B 0,C 180,E1 -29469.127,E2 -29469.127} C_VEL
LIN {X 0,Y 47.717,Z 537.312,A -85,B 0,C 180,E1 -29477.408,E2 -29477.408} C_VEL
LIN {X 0,Y 55.588,Z 537.707,A -85,B 0,C 180,E1 -29489.623,E2 -29489.623} C_VEL
LIN {X 0,Y 61.65,Z 537.219,A -85,B 0,C 180,E1 -29495.756,E2 -29495.756} C_VEL
LIN {X 0,Y 71.841,Z 535.319,A -85,B 0,C 180,E1 -29502.935,E2 -29502.935} C_VEL
LIN {X 0,Y 82.566,Z 532.122,A -85,B 0,C 180,E1 -29508.164,E2 -29508.164} C_VEL
LIN {X 0,Y 92.325,Z 528.148,A -85,B 0,C 180,E1 -29511.674,E2 -29511.674} C_VEL
LIN {X 0,Y 104.05,Z 521.911,A -85,B 0,C 180,E1 -29514.98,E2 -29514.98} C_VEL
LIN {X 0,Y 114.32,Z 515.003,A -85,B 0,C 180,E1 -29517.295,E2 -29517.295} C_VEL
LIN {X 0,Y 123.003,Z 507.909,A -85,B 0,C 180,E1 -29518.846,E2 -29518.846} C_VEL
LIN {X 0,Y 132.45,Z 498.528,A -85,B 0,C 180,E1 -29520.338,E2 -29520.338} C_VEL
LIN {X 0,Y 140.594,Z 488.519,A -85,B 0,C 180,E1 -29521.466,E2 -29521.466} C_VEL
LIN {X 0,Y 147.7,Z 477.754,A -85,B 0,C 180,E1 -29522.352,E2 -29522.352} C_VEL
LIN {X 0,Y 153.807,Z 466.064,A -85,B 0,C 180,E1 -29523.11,E2 -29523.11} C_VEL
LIN {X 0,Y 155.658,Z 461.766,A -85,B 0,C 180,E1 -29523.434,E2 -29523.434} C_VEL
LIN {X 0,Y 155.856,Z 460.772,A -85,B 0,C 180,E1 -29525.175,E2 -29525.175} C_VEL
LIN {X 0,Y 155.906,Z 460.55,A -85,B 0,C 180,E1 -29527.773,E2 -29527.773} C_VEL
LIN {X 0,Y 155.787,Z 461.687,A -85,B 0,C 180,E1 -29530.397,E2 -29530.397} C_VEL
LIN {X 0,Y 155.327,Z 463.099,A -85,B 0,C 180,E1 -29531.107,E2 -29531.107} C_VEL
LIN {X 0,Y 149.762,Z 474.69,A -85,B 0,C 180,E1 -29531.611,E2 -29531.611} C_VEL
LIN {X 0,Y 142.914,Z 485.917,A -85,B 0,C 180,E1 -29532.233,E2 -29532.233} C_VEL
LIN {X 0,Y 136.101,Z 495.014,A -85,B 0,C 180,E1 -29532.945,E2 -29532.945} C_VEL
LIN {X 0,Y 128.482,Z 503.517,A -85,B 0,C 180,E1 -29533.872,E2 -29533.872} C_VEL
LIN {X 0,Y 121.773,Z 509.892,A -85,B 0,C 180,E1 -29534.848,E2 -29534.848} C_VEL
LIN {X 0,Y 113.447,Z 516.679,A -85,B 0,C 180,E1 -29536.237,E2 -29536.237} C_VEL
LIN {X 0,Y 103.576,Z 523.372,A -85,B 0,C 180,E1 -29538.224,E2 -29538.224} C_VEL
LIN {X 0,Y 93.858,Z 528.746,A -85,B 0,C 180,E1 -29540.632,E2 -29540.632} C_VEL
LIN {X 0,Y 84.397,Z 532.97,A -85,B 0,C 180,E1 -29543.671,E2 -29543.671} C_VEL
LIN {X 0,Y 72.971,Z 536.882,A -85,B 0,C 180,E1 -29548.789,E2 -29548.789} C_VEL
LIN {X 0,Y 66.745,Z 538.426,A -85,B 0,C 180,E1 -29552.626,E2 -29552.626} C_VEL
LIN {X 0,Y 56.319,Z 540.066,A -85,B 0,C 180,E1 -29561.536,E2 -29561.536} C_VEL
LIN {X 0,Y 51.76,Z 540.313,A -85,B 0,C 180,E1 -29567.259,E2 -29567.259} C_VEL
LIN {X 0,Y 44.906,Z 539.624,A -85,B 0,C 180,E1 -29582.013,E2 -29582.013} C_VEL
LIN {X 0,Y 41.725,Z 537.425,A -85,B 0,C 180,E1 -29600.318,E2 -29600.318} C_VEL
LIN {X 0,Y 41.536,Z 535.668,A -85,B 0,C 180,E1 -29610.014,E2 -29610.014} C_VEL
LIN {X 0,Y 42.039,Z 532.103,A -85,B 0,C 180,E1 -29624.537,E2 -29624.537} C_VEL
LIN {X 0,Y 44.678,Z 527.374,A -85,B 0,C 180,E1 -29638.173,E2 -29638.173} C_VEL
LIN {X 0,Y 49.486,Z 521.368,A -85,B 0,C 180,E1 -29649.739,E2 -29649.739} C_VEL
LIN {X 0,Y 55.81,Z 513.845,A -85,B 0,C 180,E1 -29659.091,E2 -29659.091} C_VEL
LIN {X 0,Y 60.574,Z 507.778,A -85,B 0,C 180,E1 -29664.323,E2 -29664.323} C_VEL
LIN {X 0,Y 66.02,Z 500.805,A -85,B 0,C 180,E1 -29668.405,E2 -29668.405} C_VEL
LIN {X 0,Y 72.321,Z 491.3,A -85,B 0,C 180,E1 -29672.484,E2 -29672.484} C_VEL
LIN {X 0,Y 76.695,Z 483.774,A -85,B 0,C 180,E1 -29674.827,E2 -29674.827} C_VEL
LIN {X 0,Y 82.005,Z 473.199,A -85,B 0,C 180,E1 -29677.133,E2 -29677.133} C_VEL
LIN {X 0,Y 86.649,Z 461.575,A -85,B 0,C 180,E1 -29678.885,E2 -29678.885} C_VEL
LIN {X 0,Y 90.587,Z 448.254,A -85,B 0,C 180,E1 -29680.267,E2 -29680.267} C_VEL
LIN {X 0,Y 93.031,Z 435.733,A -85,B 0,C 180,E1 -29681.104,E2 -29681.104} C_VEL
LIN {X 0,Y 95.984,Z 409.293,A -85,B 0,C 180,E1 -29682.17,E2 -29682.17} C_VEL
LIN {X 0,Y 95.763,Z 407.714,A -85,B 0,C 180,E1 -29682.728,E2 -29682.728} C_VEL
LIN {X 0,Y 93.819,Z 402.385,A -85,B 0,C 180,E1 -29686.53,E2 -29686.53} C_VEL
LIN {X 0,Y 91.936,Z 397.741,A -85,B 0,C 180,E1 -29691.049,E2 -29691.049} C_VEL
LIN {X 0,Y 90.89,Z 395.28,A -85,B 0,C 180,E1 -29694.249,E2 -29694.249} C_VEL
LIN {X 0,Y 89.78,Z 392.288,A -85,B 0,C 180,E1 -29699.158,E2 -29699.158} C_VEL
LIN {X 0,Y 89.116,Z 390.838,A -85,B 0,C 180,E1 -29704.522,E2 -29704.522} C_VEL
LIN {X 0,Y 88.999,Z 391.389,A -85,B 0,C 180,E1 -29710.326,E2 -29710.326} C_VEL
LIN {X 0,Y 89.842,Z 393.023,A -85,B 0,C 180,E1 -29717.077,E2 -29717.077} C_VEL
LIN {X 0,Y 91.371,Z 396.619,A -85,B 0,C 180,E1 -29722.985,E2 -29722.985} C_VEL
LIN {X 0,Y 93.151,Z 400.773,A -85,B 0,C 180,E1 -29727.623,E2 -29727.623} C_VEL
LIN {X 0,Y 95.294,Z 406.286,A -85,B 0,C 180,E1 -29732.01,E2 -29732.01} C_VEL
LIN {X 0,Y 95.822,Z 407.774,A -85,B 0,C 180,E1 -29732.976,E2 -29732.976} C_VEL
LIN {X 0,Y 96.161,Z 410.043,A -85,B 0,C 180,E1 -29733.784,E2 -29733.784} C_VEL
LIN {X 0,Y 96.004,Z 413.62,A -85,B 0,C 180,E1 -29734.16,E2 -29734.16} C_VEL
LIN {X 0,Y 95.125,Z 418.35,A -85,B 0,C 180,E1 -29733.834,E2 -29733.834} C_VEL
LIN {X 0,Y 94.109,Z 421.997,A -85,B 0,C 180,E1 -29733.17,E2 -29733.17} C_VEL
LIN {X 0,Y 90.861,Z 432.056,A -85,B 0,C 180,E1 -29730.835,E2 -29730.835} C_VEL
LIN {X 0,Y 89.493,Z 437.327,A -85,B 0,C 180,E1 -29730.351,E2 -29730.351} C_VEL
LIN {X 0,Y 89.269,Z 438.403,A -85,B 0,C 180,E1 -29730.379,E2 -29730.379} C_VEL
LIN {X 0,Y 86.181,Z 451.03,A -85,B 0,C 180,E1 -29731.322,E2 -29731.322} C_VEL
LIN {X 0,Y 81.695,Z 464.123,A -85,B 0,C 180,E1 -29732.978,E2 -29732.978} C_VEL
LIN {X 0,Y 76.94,Z 474.537,A -85,B 0,C 180,E1 -29734.692,E2 -29734.692} C_VEL
LIN {X 0,Y 70.917,Z 485.521,A -85,B 0,C 180,E1 -29737.538,E2 -29737.538} C_VEL
LIN {X 0,Y 64.187,Z 495.556,A -85,B 0,C 180,E1 -29741.274,E2 -29741.274} C_VEL
LIN {X 0,Y 56.517,Z 505.317,A -85,B 0,C 180,E1 -29746.834,E2 -29746.834} C_VEL
LIN {X 0,Y 49.904,Z 512.658,A -85,B 0,C 180,E1 -29753.221,E2 -29753.221} C_VEL
LIN {X 0,Y 43.073,Z 519.856,A -85,B 0,C 180,E1 -29763.325,E2 -29763.325} C_VEL
LIN {X 0,Y 38.557,Z 524.731,A -85,B 0,C 180,E1 -29774.117,E2 -29774.117} C_VEL
LIN {X 0,Y 34.945,Z 529.482,A -85,B 0,C 180,E1 -29789.983,E2 -29789.983} C_VEL
LIN {X 0,Y 33.889,Z 533.13,A -85,B 0,C 180,E1 -29808.105,E2 -29808.105} C_VEL
LIN {X 0,Y 37.555,Z 536.41,A -85,B 0,C 180,E1 -29831.538,E2 -29831.538} C_VEL
LIN {X 0,Y 43.023,Z 537.658,A -85,B 0,C 180,E1 -29844.739,E2 -29844.739} C_VEL
LIN {X 0,Y 51.158,Z 537.984,A -85,B 0,C 180,E1 -29855.663,E2 -29855.663} C_VEL
LIN {X 0,Y 58.978,Z 537.382,A -85,B 0,C 180,E1 -29862.385,E2 -29862.385} C_VEL
LIN {X 0,Y 68.873,Z 535.649,A -85,B 0,C 180,E1 -29868.225,E2 -29868.225} C_VEL
LIN {X 0,Y 81.367,Z 532.091,A -85,B 0,C 180,E1 -29873.294,E2 -29873.294} C_VEL
LIN {X 0,Y 91.545,Z 528.004,A -85,B 0,C 180,E1 -29876.281,E2 -29876.281} C_VEL
LIN {X 0,Y 103.664,Z 521.612,A -85,B 0,C 180,E1 -29879.09,E2 -29879.09} C_VEL
LIN {X 0,Y 114.21,Z 514.581,A -85,B 0,C 180,E1 -29880.997,E2 -29880.997} C_VEL
LIN {X 0,Y 123.076,Z 507.34,A -85,B 0,C 180,E1 -29882.292,E2 -29882.292} C_VEL
LIN {X 0,Y 132.421,Z 498.01,A -85,B 0,C 180,E1 -29883.495,E2 -29883.495} C_VEL
LIN {X 0,Y 140.974,Z 487.466,A -85,B 0,C 180,E1 -29884.458,E2 -29884.458} C_VEL
LIN {X 0,Y 148.189,Z 476.373,A -85,B 0,C 180,E1 -29885.217,E2 -29885.217} C_VEL
LIN {X 0,Y 152.991,Z 467.187,A -85,B 0,C 180,E1 -29885.813,E2 -29885.813} C_VEL
LIN {X 0,Y 153.031,Z 467.185,A -85,B 0,C 180,E1 -29887.92,E2 -29887.92} C_VEL
LIN {X 0,Y 152.386,Z 468.631,A -85,B 0,C 180,E1 -29888.675,E2 -29888.675} C_VEL
LIN {X 0,Y 145.911,Z 480.401,A -85,B 0,C 180,E1 -29889.131,E2 -29889.131} C_VEL
LIN {X 0,Y 138.129,Z 491.594,A -85,B 0,C 180,E1 -29889.696,E2 -29889.696} C_VEL
LIN {X 0,Y 130.394,Z 500.621,A -85,B 0,C 180,E1 -29890.407,E2 -29890.407} C_VEL
LIN {X 0,Y 120.156,Z 510.391,A -85,B 0,C 180,E1 -29891.588,E2 -29891.588} C_VEL
LIN {X 0,Y 111.674,Z 517.048,A -85,B 0,C 180,E1 -29892.745,E2 -29892.745} C_VEL
LIN {X 0,Y 101.582,Z 523.626,A -85,B 0,C 180,E1 -29894.424,E2 -29894.424} C_VEL
LIN {X 0,Y 91.599,Z 528.898,A -85,B 0,C 180,E1 -29896.475,E2 -29896.475} C_VEL
LIN {X 0,Y 81.801,Z 533.026,A -85,B 0,C 180,E1 -29899.103,E2 -29899.103} C_VEL
LIN {X 0,Y 75.424,Z 535.223,A -85,B 0,C 180,E1 -29901.306,E2 -29901.306} C_VEL
LIN {X 0,Y 63.189,Z 538.306,A -85,B 0,C 180,E1 -29907.177,E2 -29907.177} C_VEL
LIN {X 0,Y 51.88,Z 539.858,A -85,B 0,C 180,E1 -29915.65,E2 -29915.65} C_VEL
LIN {X 0,Y 42.325,Z 539.824,A -85,B 0,C 180,E1 -29928.399,E2 -29928.399} C_VEL
LIN {X 0,Y 36.152,Z 538.308,A -85,B 0,C 180,E1 -29947.138,E2 -29947.138} C_VEL
LIN {X 0,Y 34.737,Z 536.947,A -85,B 0,C 180,E1 -29958.345,E2 -29958.345} C_VEL
LIN {X 0,Y 34.433,Z 535.128,A -85,B 0,C 180,E1 -29970.017,E2 -29970.017} C_VEL
LIN {X 0,Y 35.192,Z 531.469,A -85,B 0,C 180,E1 -29987.448,E2 -29987.448} C_VEL
LIN {X 0,Y 38.537,Z 526.639,A -85,B 0,C 180,E1 -30003.187,E2 -30003.187} C_VEL
LIN {X 0,Y 44.236,Z 520.523,A -85,B 0,C 180,E1 -30015.657,E2 -30015.657} C_VEL
LIN {X 0,Y 51.409,Z 512.874,A -85,B 0,C 180,E1 -30025.13,E2 -30025.13} C_VEL
LIN {X 0,Y 56.735,Z 506.676,A -85,B 0,C 180,E1 -30030.146,E2 -30030.146} C_VEL
LIN {X 0,Y 62.556,Z 499.519,A -85,B 0,C 180,E1 -30034.018,E2 -30034.018} C_VEL
LIN {X 0,Y 69.29,Z 489.804,A -85,B 0,C 180,E1 -30037.771,E2 -30037.771} C_VEL
LIN {X 0,Y 75.51,Z 479.191,A -85,B 0,C 180,E1 -30040.476,E2 -30040.476} C_VEL
LIN {X 0,Y 80.267,Z 469.284,A -85,B 0,C 180,E1 -30042.234,E2 -30042.234} C_VEL
LIN {X 0,Y 84.728,Z 457.798,A -85,B 0,C 180,E1 -30043.575,E2 -30043.575} C_VEL
LIN {X 0,Y 88.434,Z 444.267,A -85,B 0,C 180,E1 -30044.691,E2 -30044.691} C_VEL
LIN {X 0,Y 90.609,Z 431.764,A -85,B 0,C 180,E1 -30045.315,E2 -30045.315} C_VEL
LIN {X 0,Y 92.865,Z 411.641,A -85,B 0,C 180,E1 -30046.076,E2 -30046.076} C_VEL
LIN {X 0,Y 91.223,Z 406.525,A -85,B 0,C 180,E1 -30050.157,E2 -30050.157} C_VEL
LIN {X 0,Y 89.733,Z 402.325,A -85,B 0,C 180,E1 -30054.944,E2 -30054.944} C_VEL
LIN {X 0,Y 88.635,Z 399.046,A -85,B 0,C 180,E1 -30060.533,E2 -30060.533} C_VEL
LIN {X 0,Y 88.229,Z 397.889,A -85,B 0,C 180,E1 -30064.568,E2 -30064.568} C_VEL
LIN {X 0,Y 88.094,Z 398.386,A -85,B 0,C 180,E1 -30069.806,E2 -30069.806} C_VEL
LIN {X 0,Y 88.699,Z 399.793,A -85,B 0,C 180,E1 -30075.838,E2 -30075.838} C_VEL
LIN {X 0,Y 89.935,Z 403.203,A -85,B 0,C 180,E1 -30081.526,E2 -30081.526} C_VEL
LIN {X 0,Y 91.335,Z 406.999,A -85,B 0,C 180,E1 -30085.799,E2 -30085.799} C_VEL
LIN {X 0,Y 92.76,Z 411.258,A -85,B 0,C 180,E1 -30089.293,E2 -30089.293} C_VEL
LIN {X 0,Y 90.019,Z 434.225,A -85,B 0,C 180,E1 -30090.168,E2 -30090.168} C_VEL
LIN {X 0,Y 89.269,Z 438.403,A -85,B 0,C 180,E1 -30090.379,E2 -30090.379} C_VEL
LIN {X 0,Y 87.784,Z 444.135,A -85,B 0,C 180,E1 -30090.323,E2 -30090.323} C_VEL
LIN {X 0,Y 84.244,Z 453.29,A -85,B 0,C 180,E1 -30089.311,E2 -30089.311} C_VEL
LIN {X 0,Y 80.08,Z 462.192,A -85,B 0,C 180,E1 -30088.458,E2 -30088.458} C_VEL
LIN {X 0,Y 77.581,Z 467.521,A -85,B 0,C 180,E1 -30088.754,E2 -30088.754} C_VEL
LIN {X 0,Y 71.515,Z 479.338,A -85,B 0,C 180,E1 -30090.68,E2 -30090.68} C_VEL
LIN {X 0,Y 64.489,Z 490.507,A -85,B 0,C 180,E1 -30093.714,E2 -30093.714} C_VEL
LIN {X 0,Y 56.683,Z 500.632,A -85,B 0,C 180,E1 -30097.907,E2 -30097.907} C_VEL
LIN {X 0,Y 48.621,Z 509.486,A -85,B 0,C 180,E1 -30103.702,E2 -30103.702} C_VEL
LIN {X 0,Y 40.434,Z 517.36,A -85,B 0,C 180,E1 -30112.512,E2 -30112.512} C_VEL
LIN {X 0,Y 33.577,Z 523.652,A -85,B 0,C 180,E1 -30125.233,E2 -30125.233} C_VEL
LIN {X 0,Y 29.052,Z 528.269,A -85,B 0,C 180,E1 -30141.097,E2 -30141.097} C_VEL
LIN {X 0,Y 26.754,Z 532.588,A -85,B 0,C 180,E1 -30165.206,E2 -30165.206} C_VEL
LIN {X 0,Y 27.69,Z 534.615,A -85,B 0,C 180,E1 -30180.48,E2 -30180.48} C_VEL
LIN {X 0,Y 31.659,Z 536.625,A -85,B 0,C 180,E1 -30198.247,E2 -30198.247} C_VEL
LIN {X 0,Y 39.192,Z 538.004,A -85,B 0,C 180,E1 -30213.679,E2 -30213.679} C_VEL
LIN {X 0,Y 47.416,Z 538.261,A -85,B 0,C 180,E1 -30222.758,E2 -30222.758} C_VEL
LIN {X 0,Y 57.162,Z 537.545,A -85,B 0,C 180,E1 -30229.545,E2 -30229.545} C_VEL
LIN {X 0,Y 66.515,Z 535.985,A -85,B 0,C 180,E1 -30233.936,E2 -30233.936} C_VEL
LIN {X 0,Y 77.364,Z 533.15,A -85,B 0,C 180,E1 -30237.608,E2 -30237.608} C_VEL
LIN {X 0,Y 86.877,Z 529.743,A -85,B 0,C 180,E1 -30240.001,E2 -30240.001} C_VEL
LIN {X 0,Y 98.459,Z 524.326,A -85,B 0,C 180,E1 -30242.292,E2 -30242.292} C_VEL
LIN {X 0,Y 109.63,Z 517.642,A -85,B 0,C 180,E1 -30244.063,E2 -30244.063} C_VEL
LIN {X 0,Y 119.982,Z 509.836,A -85,B 0,C 180,E1 -30245.327,E2 -30245.327} C_VEL
LIN {X 0,Y 128.995,Z 501.524,A -85,B 0,C 180,E1 -30246.268,E2 -30246.268} C_VEL
LIN {X 0,Y 134.464,Z 495.639,A -85,B 0,C 180,E1 -30246.794,E2 -30246.794} C_VEL
LIN {X 0,Y 134.51,Z 495.597,A -85,B 0,C 180,E1 -30246.958,E2 -30246.958} C_VEL
LIN {X 0,Y 125.846,Z 504.719,A -85,B 0,C 180,E1 -30247.621,E2 -30247.621} C_VEL
LIN {X 0,Y 117.224,Z 512.27,A -85,B 0,C 180,E1 -30248.455,E2 -30248.455} C_VEL
LIN {X 0,Y 110.328,Z 517.418,A -85,B 0,C 180,E1 -30249.158,E2 -30249.158} C_VEL
LIN {X 0,Y 100.053,Z 523.879,A -85,B 0,C 180,E1 -30250.49,E2 -30250.49} C_VEL
LIN {X 0,Y 89.842,Z 529.043,A -85,B 0,C 180,E1 -30252.124,E2 -30252.124} C_VEL
LIN {X 0,Y 79.76,Z 533.079,A -85,B 0,C 180,E1 -30254.278,E2 -30254.278} C_VEL
LIN {X 0,Y 73.136,Z 535.189,A -85,B 0,C 180,E1 -30256.098,E2 -30256.098} C_VEL
LIN {X 0,Y 60.263,Z 538.186,A -85,B 0,C 180,E1 -30261.125,E2 -30261.125} C_VEL
LIN {X 0,Y 54.042,Z 539.109,A -85,B 0,C 180,E1 -30264.477,E2 -30264.477} C_VEL
LIN {X 0,Y 42.435,Z 539.744,A -85,B 0,C 180,E1 -30274.123,E2 -30274.123} C_VEL
LIN {X 0,Y 32.985,Z 538.885,A -85,B 0,C 180,E1 -30290.291,E2 -30290.291} C_VEL
LIN {X 0,Y 29.736,Z 537.888,A -85,B 0,C 180,E1 -30301.815,E2 -30301.815} C_VEL
LIN {X 0,Y 27.822,Z 536.451,A -85,B 0,C 180,E1 -30315.391,E2 -30315.391} C_VEL
LIN {X 0,Y 27.349,Z 534.589,A -85,B 0,C 180,E1 -30330.022,E2 -30330.022} C_VEL
LIN {X 0,Y 28.462,Z 530.833,A -85,B 0,C 180,E1 -30351.762,E2 -30351.762} C_VEL
LIN {X 0,Y 32.788,Z 525.902,A -85,B 0,C 180,E1 -30370.042,E2 -30370.042} C_VEL
LIN {X 0,Y 39.579,Z 519.679,A -85,B 0,C 180,E1 -30383.064,E2 -30383.064} C_VEL
LIN {X 0,Y 47.664,Z 511.868,A -85,B 0,C 180,E1 -30392.239,E2 -30392.239} C_VEL
LIN {X 0,Y 52.364,Z 506.83,A -85,B 0,C 180,E1 -30396.046,E2 -30396.046} C_VEL
LIN {X 0,Y 59.765,Z 498.235,A -85,B 0,C 180,E1 -30400.207,E2 -30400.207} C_VEL
LIN {X 0,Y 66.094,Z 489.497,A -85,B 0,C 180,E1 -30403.165,E2 -30403.165} C_VEL
LIN {X 0,Y 72.612,Z 478.889,A -85,B 0,C 180,E1 -30405.471,E2 -30405.471} C_VEL
LIN {X 0,Y 78.391,Z 467.108,A -85,B 0,C 180,E1 -30407.186,E2 -30407.186} C_VEL
LIN {X 0,Y 82.741,Z 455.665,A -85,B 0,C 180,E1 -30408.243,E2 -30408.243} C_VEL
LIN {X 0,Y 86.327,Z 442.387,A -85,B 0,C 180,E1 -30409.132,E2 -30409.132} C_VEL
LIN {X 0,Y 88.557,Z 428.749,A -85,B 0,C 180,E1 -30409.653,E2 -30409.653} C_VEL
LIN {X 0,Y 90.109,Z 414.858,A -85,B 0,C 180,E1 -30410.2,E2 -30410.2} C_VEL
LIN {X 0,Y 88.818,Z 410.384,A -85,B 0,C 180,E1 -30414.607,E2 -30414.607} C_VEL
LIN {X 0,Y 87.971,Z 407.693,A -85,B 0,C 180,E1 -30418.568,E2 -30418.568} C_VEL
LIN {X 0,Y 87.584,Z 405.876,A -85,B 0,C 180,E1 -30421.619,E2 -30421.619} C_VEL
LIN {X 0,Y 87.332,Z 405.024,A -85,B 0,C 180,E1 -30424.615,E2 -30424.615} C_VEL
LIN {X 0,Y 87.197,Z 405.384,A -85,B 0,C 180,E1 -30429.275,E2 -30429.275} C_VEL
LIN {X 0,Y 87.661,Z 406.879,A -85,B 0,C 180,E1 -30435.123,E2 -30435.123} C_VEL
LIN {X 0,Y 88.588,Z 409.917,A -85,B 0,C 180,E1 -30440.155,E2 -30440.155} C_VEL
LIN {X 0,Y 89.633,Z 413.421,A -85,B 0,C 180,E1 -30443.999,E2 -30443.999} C_VEL
LIN {X 0,Y 89.992,Z 414.649,A -85,B 0,C 180,E1 -30445.115,E2 -30445.115} C_VEL
LIN {X 0,Y 87.664,Z 433.939,A -85,B 0,C 180,E1 -30445.858,E2 -30445.858} C_VEL
LIN {X 0,Y 84.848,Z 446.907,A -85,B 0,C 180,E1 -30446.551,E2 -30446.551} C_VEL
LIN {X 0,Y 80.819,Z 459.63,A -85,B 0,C 180,E1 -30447.739,E2 -30447.739} C_VEL
LIN {X 0,Y 77.581,Z 467.521,A -85,B 0,C 180,E1 -30448.754,E2 -30448.754} C_VEL
LIN {X 0,Y 74.845,Z 472.832,A -85,B 0,C 180,E1 -30449.108,E2 -30449.108} C_VEL
LIN {X 0,Y 69.32,Z 481.067,A -85,B 0,C 180,E1 -30448.409,E2 -30448.409} C_VEL
LIN {X 0,Y 63.266,Z 488.86,A -85,B 0,C 180,E1 -30447.785,E2 -30447.785} C_VEL
LIN {X 0,Y 59.684,Z 493.413,A -85,B 0,C 180,E1 -30448.494,E2 -30448.494} C_VEL
LIN {X 0,Y 52.03,Z 502.505,A -85,B 0,C 180,E1 -30452.028,E2 -30452.028} C_VEL
LIN {X 0,Y 43.98,Z 510.552,A -85,B 0,C 180,E1 -30456.944,E2 -30456.944} C_VEL
LIN {X 0,Y 35.014,Z 518.241,A -85,B 0,C 180,E1 -30465.347,E2 -30465.347} C_VEL
LIN {X 0,Y 27.217,Z 524.418,A -85,B 0,C 180,E1 -30478.881,E2 -30478.881} C_VEL
LIN {X 0,Y 21.304,Z 529.539,A -85,B 0,C 180,E1 -30501.729,E2 -30501.729} C_VEL
LIN {X 0,Y 19.739,Z 533.163,A -85,B 0,C 180,E1 -30530.825,E2 -30530.825} C_VEL
LIN {X 0,Y 21.661,Z 535.139,A -85,B 0,C 180,E1 -30550.423,E2 -30550.423} C_VEL
LIN {X 0,Y 26.41,Z 536.844,A -85,B 0,C 180,E1 -30567.847,E2 -30567.847} C_VEL
LIN {X 0,Y 36.503,Z 538.351,A -85,B 0,C 180,E1 -30584.229,E2 -30584.229} C_VEL
LIN {X 0,Y 44.501,Z 538.538,A -85,B 0,C 180,E1 -30590.915,E2 -30590.915} C_VEL
LIN {X 0,Y 56.287,Z 537.709,A -85,B 0,C 180,E1 -30597.05,E2 -30597.05} C_VEL
LIN {X 0,Y 64.914,Z 536.31,A -85,B 0,C 180,E1 -30600.001,E2 -30600.001} C_VEL
LIN {X 0,Y 77.412,Z 533.123,A -85,B 0,C 180,E1 -30603.129,E2 -30603.129} C_VEL
LIN {X 0,Y 88.417,Z 529.12,A -85,B 0,C 180,E1 -30605.08,E2 -30605.08} C_VEL
LIN {X 0,Y 95.701,Z 525.794,A -85,B 0,C 180,E1 -30606.156,E2 -30606.156} C_VEL
LIN {X 0,Y 92.083,Z 527.58,A -85,B 0,C 180,E1 -30607.221,E2 -30607.221} C_VEL
LIN {X 0,Y 81.736,Z 531.885,A -85,B 0,C 180,E1 -30608.628,E2 -30608.628} C_VEL
LIN {X 0,Y 71.494,Z 535.154,A -85,B 0,C 180,E1 -30610.622,E2 -30610.622} C_VEL
LIN {X 0,Y 58.073,Z 538.066,A -85,B 0,C 180,E1 -30614.541,E2 -30614.541} C_VEL
LIN {X 0,Y 51.503,Z 538.924,A -85,B 0,C 180,E1 -30617.257,E2 -30617.257} C_VEL
LIN {X 0,Y 38.899,Z 539.458,A -85,B 0,C 180,E1 -30625.433,E2 -30625.433} C_VEL
LIN {X 0,Y 27.875,Z 538.513,A -85,B 0,C 180,E1 -30640.888,E2 -30640.888} C_VEL
LIN {X 0,Y 23.695,Z 537.438,A -85,B 0,C 180,E1 -30653.648,E2 -30653.648} C_VEL
LIN {X 0,Y 21.04,Z 535.957,A -85,B 0,C 180,E1 -30670.517,E2 -30670.517} C_VEL
LIN {X 0,Y 20.247,Z 534.05,A -85,B 0,C 180,E1 -30690.03,E2 -30690.03} C_VEL
LIN {X 0,Y 22.005,Z 530.199,A -85,B 0,C 180,E1 -30718.655,E2 -30718.655} C_VEL
LIN {X 0,Y 27.689,Z 525.165,A -85,B 0,C 180,E1 -30739.625,E2 -30739.625} C_VEL
LIN {X 0,Y 35.742,Z 518.83,A -85,B 0,C 180,E1 -30752.266,E2 -30752.266} C_VEL
LIN {X 0,Y 44.756,Z 510.818,A -85,B 0,C 180,E1 -30760.457,E2 -30760.457} C_VEL
LIN {X 0,Y 50.073,Z 505.554,A -85,B 0,C 180,E1 -30763.605,E2 -30763.605} C_VEL
LIN {X 0,Y 57.725,Z 496.946,A -85,B 0,C 180,E1 -30766.949,E2 -30766.949} C_VEL
LIN {X 0,Y 64.376,Z 487.998,A -85,B 0,C 180,E1 -30769.324,E2 -30769.324} C_VEL
LIN {X 0,Y 71.163,Z 477.095,A -85,B 0,C 180,E1 -30771.014,E2 -30771.014} C_VEL
LIN {X 0,Y 76.267,Z 466.786,A -85,B 0,C 180,E1 -30772.197,E2 -30772.197} C_VEL
LIN {X 0,Y 81.032,Z 454.404,A -85,B 0,C 180,E1 -30773.054,E2 -30773.054} C_VEL
LIN {X 0,Y 84.607,Z 441.202,A -85,B 0,C 180,E1 -30773.718,E2 -30773.718} C_VEL
LIN {X 0,Y 86.885,Z 426.671,A -85,B 0,C 180,E1 -30774.165,E2 -30774.165} C_VEL
LIN {X 0,Y 87.836,Z 418.64,A -85,B 0,C 180,E1 -30774.391,E2 -30774.391} C_VEL
LIN {X 0,Y 86.981,Z 415,A -85,B 0,C 180,E1 -30778.842,E2 -30778.842} C_VEL
LIN {X 0,Y 86.502,Z 412.553,A -85,B 0,C 180,E1 -30783.422,E2 -30783.422} C_VEL
LIN {X 0,Y 86.355,Z 412.065,A -85,B 0,C 180,E1 -30786.281,E2 -30786.281} C_VEL
LIN {X 0,Y 86.558,Z 413.412,A -85,B 0,C 180,E1 -30793.435,E2 -30793.435} C_VEL
LIN {X 0,Y 87.332,Z 416.748,A -85,B 0,C 180,E1 -30798.929,E2 -30798.929} C_VEL
LIN {X 0,Y 87.738,Z 418.418,A -85,B 0,C 180,E1 -30800.856,E2 -30800.856} C_VEL
LIN {X 0,Y 85.656,Z 434.563,A -85,B 0,C 180,E1 -30801.351,E2 -30801.351} C_VEL
LIN {X 0,Y 82.73,Z 447.548,A -85,B 0,C 180,E1 -30801.923,E2 -30801.923} C_VEL
LIN {X 0,Y 78.536,Z 460.28,A -85,B 0,C 180,E1 -30802.918,E2 -30802.918} C_VEL
LIN {X 0,Y 73.211,Z 472.132,A -85,B 0,C 180,E1 -30804.204,E2 -30804.204} C_VEL
LIN {X 0,Y 67.343,Z 482.437,A -85,B 0,C 180,E1 -30805.808,E2 -30805.808} C_VEL
LIN {X 0,Y 61.84,Z 490.609,A -85,B 0,C 180,E1 -30807.747,E2 -30807.747} C_VEL
LIN {X 0,Y 59.684,Z 493.413,A -85,B 0,C 180,E1 -30808.494,E2 -30808.494} C_VEL
LIN {X 0,Y 55.921,Z 497.895,A -85,B 0,C 180,E1 -30809.379,E2 -30809.379} C_VEL
LIN {X 0,Y 48.742,Z 504.775,A -85,B 0,C 180,E1 -30809.202,E2 -30809.202} C_VEL
LIN {X 0,Y 41.011,Z 511.049,A -85,B 0,C 180,E1 -30809.15,E2 -30809.15} C_VEL
LIN {X 0,Y 36.402,Z 514.585,A -85,B 0,C 180,E1 -30810.912,E2 -30810.912} C_VEL
LIN {X 0,Y 27.236,Z 521.297,A -85,B 0,C 180,E1 -30819.242,E2 -30819.242} C_VEL
LIN {X 0,Y 18.7,Z 526.916,A -85,B 0,C 180,E1 -30835.648,E2 -30835.648} C_VEL
LIN {X 0,Y 12.993,Z 531.365,A -85,B 0,C 180,E1 -30869.954,E2 -30869.954} C_VEL
LIN {X 0,Y 13.137,Z 533.737,A -85,B 0,C 180,E1 -30902.288,E2 -30902.288} C_VEL
LIN {X 0,Y 16.745,Z 535.631,A -85,B 0,C 180,E1 -30927.01,E2 -30927.01} C_VEL
LIN {X 0,Y 22.214,Z 537.059,A -85,B 0,C 180,E1 -30941.56,E2 -30941.56} C_VEL
LIN {X 0,Y 28.501,Z 538.083,A -85,B 0,C 180,E1 -30950.397,E2 -30950.397} C_VEL
LIN {X 0,Y 35.217,Z 538.684,A -85,B 0,C 180,E1 -30955.943,E2 -30955.943} C_VEL
LIN {X 0,Y 42.673,Z 538.814,A -85,B 0,C 180,E1 -30960.002,E2 -30960.002} C_VEL
LIN {X 0,Y 56.397,Z 537.872,A -85,B 0,C 180,E1 -30964.633,E2 -30964.633} C_VEL
LIN {X 0,Y 60.447,Z 537.31,A -85,B 0,C 180,E1 -30966.678,E2 -30966.678} C_VEL
LIN {X 0,Y 49.858,Z 538.721,A -85,B 0,C 180,E1 -30969.428,E2 -30969.428} C_VEL
LIN {X 0,Y 36.411,Z 539.172,A -85,B 0,C 180,E1 -30975.248,E2 -30975.248} C_VEL
LIN {X 0,Y 29.919,Z 538.841,A -85,B 0,C 180,E1 -30980.073,E2 -30980.073} C_VEL
LIN {X 0,Y 23.83,Z 538.115,A -85,B 0,C 180,E1 -30987.834,E2 -30987.834} C_VEL
LIN {X 0,Y 14.538,Z 535.462,A -85,B 0,C 180,E1 -31021.138,E2 -31021.138} C_VEL
LIN {X 0,Y 13.16,Z 533.512,A -85,B 0,C 180,E1 -31050.046,E2 -31050.046} C_VEL
LIN {X 0,Y 16.103,Z 529.563,A -85,B 0,C 180,E1 -31090.943,E2 -31090.943} C_VEL
LIN {X 0,Y 25.17,Z 523.421,A -85,B 0,C 180,E1 -31115.211,E2 -31115.211} C_VEL
LIN {X 0,Y 34.634,Z 516.684,A -85,B 0,C 180,E1 -31124.616,E2 -31124.616} C_VEL
LIN {X 0,Y 44.174,Z 508.585,A -85,B 0,C 180,E1 -31130.291,E2 -31130.291} C_VEL
LIN {X 0,Y 51.404,Z 501.486,A -85,B 0,C 180,E1 -31132.49,E2 -31132.49} C_VEL
LIN {X 0,Y 59.994,Z 491.296,A -85,B 0,C 180,E1 -31134.811,E2 -31134.811} C_VEL
LIN {X 0,Y 65.177,Z 483.858,A -85,B 0,C 180,E1 -31135.999,E2 -31135.999} C_VEL
LIN {X 0,Y 72.141,Z 471.924,A -85,B 0,C 180,E1 -31137.061,E2 -31137.061} C_VEL
LIN {X 0,Y 77.833,Z 459.039,A -85,B 0,C 180,E1 -31137.815,E2 -31137.815} C_VEL
